LIN {X 0,Y 365.856,Z 163.635,A -85,B 0,C 180,E1 -13024.033,E2 -13024.033} C_VEL
LIN {X 0,Y 364.238,Z 181.611,A -85,B 0,C 180,E1 -13027.845,E2 -13027.845} C_VEL
LIN {X 0,Y 364.107,Z 184.215,A -85,B 0,C 180,E1 -13028.356,E2 -13028.356} C_VEL
LIN {X 0,Y 369.085,Z 220.666,A -85,B 0,C 180,E1 -13029.411,E2 -13029.411} C_VEL
LIN {X 0,Y 367.83,Z 293.633,A -85,B 0,C 180,E1 -13030.937,E2 -13030.937} C_VEL
LIN {X 0,Y 367.143,Z 307.184,A -85,B 0,C 180,E1 -13031.443,E2 -13031.443} C_VEL
LIN {X 0,Y 366.249,Z 319.505,A -85,B 0,C 180,E1 -13032.12,E2 -13032.12} C_VEL
LIN {X 0,Y 365.195,Z 332.175,A -85,B 0,C 180,E1 -13033.078,E2 -13033.078} C_VEL
LIN {X 0,Y 364.123,Z 343.479,A -85,B 0,C 180,E1 -13034.179,E2 -13034.179} C_VEL
LIN {X 0,Y 363.21,Z 353.677,A -85,B 0,C 180,E1 -13035.431,E2 -13035.431} C_VEL
LIN {X 0,Y 362.33,Z 362.875,A -85,B 0,C 180,E1 -13036.826,E2 -13036.826} C_VEL
LIN {X 0,Y 361.664,Z 370.474,A -85,B 0,C 180,E1 -13038.227,E2 -13038.227} C_VEL
LIN {X 0,Y 361.049,Z 377.925,A -85,B 0,C 180,E1 -13039.91,E2 -13039.91} C_VEL
LIN {X 0,Y 360.671,Z 383.894,A -85,B 0,C 180,E1 -13041.596,E2 -13041.596} C_VEL
LIN {X 0,Y 360.485,Z 388.587,A -85,B 0,C 180,E1 -13043.282,E2 -13043.282} C_VEL
LIN {X 0,Y 360.383,Z 392.138,A -85,B 0,C 180,E1 -13044.965,E2 -13044.965} C_VEL
LIN {X 0,Y 360.391,Z 394.652,A -85,B 0,C 180,E1 -13046.646,E2 -13046.646} C_VEL
LIN {X 0,Y 360.472,Z 395.803,A -85,B 0,C 180,E1 -13047.765,E2 -13047.765} C_VEL
LIN {X 0,Y 360.534,Z 396.505,A -85,B 0,C 180,E1 -13048.883,E2 -13048.883} C_VEL
LIN {X 0,Y 360.52,Z 396.804,A -85,B 0,C 180,E1 -13050,E2 -13050} C_VEL
LIN {X 0,Y 360.522,Z 396.707,A -85,B 0,C 180,E1 -13051.117,E2 -13051.117} C_VEL
LIN {X 0,Y 360.428,Z 396.188,A -85,B 0,C 180,E1 -13052.235,E2 -13052.235} C_VEL
LIN {X 0,Y 360.403,Z 393.878,A -85,B 0,C 180,E1 -13054.474,E2 -13054.474} C_VEL
LIN {X 0,Y 360.378,Z 391.416,A -85,B 0,C 180,E1 -13055.961,E2 -13055.961} C_VEL
LIN {X 0,Y 360.596,Z 387.143,A -85,B 0,C 180,E1 -13057.841,E2 -13057.841} C_VEL
LIN {X 0,Y 360.914,Z 382.124,A -85,B 0,C 180,E1 -13059.527,E2 -13059.527} C_VEL
LIN {X 0,Y 361.455,Z 375.833,A -85,B 0,C 180,E1 -13061.212,E2 -13061.212} C_VEL
LIN {X 0,Y 362.392,Z 368.049,A -85,B 0,C 180,E1 -13062.887,E2 -13062.887} C_VEL
LIN {X 0,Y 363.271,Z 360.101,A -85,B 0,C 180,E1 -13064.28,E2 -13064.28} C_VEL
LIN {X 0,Y 364.321,Z 350.431,A -85,B 0,C 180,E1 -13065.668,E2 -13065.668} C_VEL
LIN {X 0,Y 365.477,Z 339.745,A -85,B 0,C 180,E1 -13066.909,E2 -13066.909} C_VEL
LIN {X 0,Y 366.789,Z 327.812,A -85,B 0,C 180,E1 -13067.997,E2 -13067.997} C_VEL
LIN {X 0,Y 367.96,Z 315.104,A -85,B 0,C 180,E1 -13068.875,E2 -13068.875} C_VEL
LIN {X 0,Y 368.927,Z 302.489,A -85,B 0,C 180,E1 -13069.51,E2 -13069.51} C_VEL
LIN {X 0,Y 369.584,Z 289.242,A -85,B 0,C 180,E1 -13069.944,E2 -13069.944} C_VEL
LIN {X 0,Y 370.844,Z 219.661,A -85,B 0,C 180,E1 -13071.411,E2 -13071.411} C_VEL
LIN {X 0,Y 367.604,Z 196.928,A -85,B 0,C 180,E1 -13072.15,E2 -13072.15} C_VEL
LIN {X 0,Y 364.788,Z 182.019,A -85,B 0,C 180,E1 -13072.701,E2 -13072.701} C_VEL
LIN {X 0,Y 366.272,Z 167.518,A -85,B 0,C 180,E1 -13075.777,E2 -13075.777} C_VEL
LIN {X 0,Y 366.461,Z 164.278,A -85,B 0,C 180,E1 -13076.48,E2 -13076.48} C_VEL
LIN {X 0,Y 364.559,Z 154.623,A -85,B 0,C 180,E1 -13078.813,E2 -13078.813} C_VEL
LIN {X 0,Y 361.909,Z 143.406,A -85,B 0,C 180,E1 -13081.704,E2 -13081.704} C_VEL
LIN {X 0,Y 361.869,Z 143.411,A -85,B 0,C 180,E1 -13085.636,E2 -13085.636} C_VEL
LIN {X 0,Y 361.875,Z 143.411,A -85,B 0,C 180,E1 -13089.027,E2 -13089.027} C_VEL
LIN {X 0,Y 361.857,Z 143.415,A -85,B 0,C 180,E1 -13092.435,E2 -13092.435} C_VEL
LIN {X 0,Y 361.826,Z 143.416,A -85,B 0,C 180,E1 -13095.945,E2 -13095.945} C_VEL
LIN {X 0,Y 361.872,Z 143.408,A -85,B 0,C 180,E1 -13099.237,E2 -13099.237} C_VEL
LIN {X 0,Y 361.869,Z 143.408,A -85,B 0,C 180,E1 -13102.982,E2 -13102.982} C_VEL
LIN {X 0,Y 361.858,Z 143.406,A -85,B 0,C 180,E1 -13106.63,E2 -13106.63} C_VEL
LIN {X 0,Y 361.874,Z 143.406,A -85,B 0,C 180,E1 -13109.672,E2 -13109.672} C_VEL
LIN {X 0,Y 361.953,Z 143.394,A -85,B 0,C 180,E1 -13113.475,E2 -13113.475} C_VEL
LIN {X 0,Y 361.881,Z 143.402,A -85,B 0,C 180,E1 -13117.144,E2 -13117.144} C_VEL
LIN {X 0,Y 361.919,Z 143.396,A -85,B 0,C 180,E1 -13120.724,E2 -13120.724} C_VEL
LIN {X 0,Y 361.945,Z 143.393,A -85,B 0,C 180,E1 -13124.226,E2 -13124.226} C_VEL
LIN {X 0,Y 361.997,Z 143.391,A -85,B 0,C 180,E1 -13126.528,E2 -13126.528} C_VEL
LIN {X 0,Y 362.03,Z 143.388,A -85,B 0,C 180,E1 -13129.938,E2 -13129.938} C_VEL
LIN {X 0,Y 362.15,Z 143.368,A -85,B 0,C 180,E1 -13132.192,E2 -13132.192} C_VEL
LIN {X 0,Y 362.117,Z 143.377,A -85,B 0,C 180,E1 -13134.431,E2 -13134.431} C_VEL
LIN {X 0,Y 362.281,Z 143.357,A -85,B 0,C 180,E1 -13137.776,E2 -13137.776} C_VEL
LIN {X 0,Y 362.426,Z 143.334,A -85,B 0,C 180,E1 -13140,E2 -13140} C_VEL
LIN {X 0,Y 362.281,Z 143.356,A -85,B 0,C 180,E1 -13142.223,E2 -13142.223} C_VEL
LIN {X 0,Y 362.159,Z 143.37,A -85,B 0,C 180,E1 -13146.686,E2 -13146.686} C_VEL
LIN {X 0,Y 362.029,Z 143.389,A -85,B 0,C 180,E1 -13150.062,E2 -13150.062} C_VEL
LIN {X 0,Y 361.996,Z 143.391,A -85,B 0,C 180,E1 -13153.899,E2 -13153.899} C_VEL
LIN {X 0,Y 361.965,Z 143.397,A -85,B 0,C 180,E1 -13157.938,E2 -13157.938} C_VEL
LIN {X 0,Y 361.89,Z 143.406,A -85,B 0,C 180,E1 -13161.653,E2 -13161.653} C_VEL
LIN {X 0,Y 361.926,Z 143.407,A -85,B 0,C 180,E1 -13165.29,E2 -13165.29} C_VEL
LIN {X 0,Y 361.93,Z 143.475,A -85,B 0,C 180,E1 -13168.883,E2 -13168.883} C_VEL
LIN {X 0,Y 362.983,Z 148.175,A -85,B 0,C 180,E1 -13170.225,E2 -13170.225} C_VEL
LIN {X 0,Y 370.942,Z 167.193,A -85,B 0,C 180,E1 -13171.263,E2 -13171.263} C_VEL
LIN {X 0,Y 371.99,Z 171.078,A -85,B 0,C 180,E1 -13171.427,E2 -13171.427} C_VEL
LIN {X 0,Y 370.044,Z 255.779,A -85,B 0,C 180,E1 -13173.22,E2 -13173.22} C_VEL
LIN {X 0,Y 369.483,Z 268.943,A -85,B 0,C 180,E1 -13173.723,E2 -13173.723} C_VEL
LIN {X 0,Y 368.876,Z 280.401,A -85,B 0,C 180,E1 -13174.362,E2 -13174.362} C_VEL
LIN {X 0,Y 368.043,Z 291.787,A -85,B 0,C 180,E1 -13175.201,E2 -13175.201} C_VEL
LIN {X 0,Y 366.955,Z 303.498,A -85,B 0,C 180,E1 -13176.32,E2 -13176.32} C_VEL
LIN {X 0,Y 365.859,Z 314.056,A -85,B 0,C 180,E1 -13177.592,E2 -13177.592} C_VEL
LIN {X 0,Y 364.797,Z 323.086,A -85,B 0,C 180,E1 -13178.937,E2 -13178.937} C_VEL
LIN {X 0,Y 363.599,Z 332.307,A -85,B 0,C 180,E1 -13180.654,E2 -13180.654} C_VEL
LIN {X 0,Y 362.718,Z 338.973,A -85,B 0,C 180,E1 -13182.198,E2 -13182.198} C_VEL
LIN {X 0,Y 361.961,Z 345.413,A -85,B 0,C 180,E1 -13184.077,E2 -13184.077} C_VEL
LIN {X 0,Y 361.32,Z 350.44,A -85,B 0,C 180,E1 -13186.028,E2 -13186.028} C_VEL
LIN {X 0,Y 360.911,Z 353.66,A -85,B 0,C 180,E1 -13187.729,E2 -13187.729} C_VEL
LIN {X 0,Y 360.497,Z 356.39,A -85,B 0,C 180,E1 -13189.959,E2 -13189.959} C_VEL
LIN {X 0,Y 360.413,Z 357.239,A -85,B 0,C 180,E1 -13191.392,E2 -13191.392} C_VEL
LIN {X 0,Y 360.34,Z 357.426,A -85,B 0,C 180,E1 -13193.097,E2 -13193.097} C_VEL
LIN {X 0,Y 360.388,Z 356.541,A -85,B 0,C 180,E1 -13194.989,E2 -13194.989} C_VEL
LIN {X 0,Y 360.584,Z 354.422,A -85,B 0,C 180,E1 -13196.939,E2 -13196.939} C_VEL
LIN {X 0,Y 360.927,Z 350.862,A -85,B 0,C 180,E1 -13198.956,E2 -13198.956} C_VEL
LIN {X 0,Y 361.405,Z 345.506,A -85,B 0,C 180,E1 -13201.055,E2 -13201.055} C_VEL
LIN {X 0,Y 361.952,Z 339.784,A -85,B 0,C 180,E1 -13202.761,E2 -13202.761} C_VEL
LIN {X 0,Y 362.663,Z 332.625,A -85,B 0,C 180,E1 -13204.458,E2 -13204.458} C_VEL
LIN {X 0,Y 363.496,Z 324.252,A -85,B 0,C 180,E1 -13206.045,E2 -13206.045} C_VEL
LIN {X 0,Y 364.462,Z 314.352,A -85,B 0,C 180,E1 -13207.561,E2 -13207.561} C_VEL
LIN {X 0,Y 365.415,Z 303.701,A -85,B 0,C 180,E1 -13208.862,E2 -13208.862} C_VEL
LIN {X 0,Y 366.4,Z 291.564,A -85,B 0,C 180,E1 -13210.031,E2 -13210.031} C_VEL
LIN {X 0,Y 367.136,Z 279.291,A -85,B 0,C 180,E1 -13210.941,E2 -13210.941} C_VEL
LIN {X 0,Y 367.783,Z 265.953,A -85,B 0,C 180,E1 -13211.657,E2 -13211.657} C_VEL
LIN {X 0,Y 368.21,Z 253.401,A -85,B 0,C 180,E1 -13212.111,E2 -13212.111} C_VEL
LIN {X 0,Y 369.689,Z 169.162,A -85,B 0,C 180,E1 -13213.858,E2 -13213.858} C_VEL
LIN {X 0,Y 367.562,Z 160.789,A -85,B 0,C 180,E1 -13214.153,E2 -13214.153} C_VEL
LIN {X 0,Y 362.572,Z 146.411,A -85,B 0,C 180,E1 -13214.766,E2 -13214.766} C_VEL
LIN {X 0,Y 361.989,Z 143.397,A -85,B 0,C 180,E1 -13215.609,E2 -13215.609} C_VEL
LIN {X 0,Y 361.969,Z 143.393,A -85,B 0,C 180,E1 -13218.804,E2 -13218.804} C_VEL
LIN {X 0,Y 362.116,Z 143.376,A -85,B 0,C 180,E1 -13222.192,E2 -13222.192} C_VEL
LIN {X 0,Y 362.114,Z 143.375,A -85,B 0,C 180,E1 -13224.431,E2 -13224.431} C_VEL
LIN {X 0,Y 362.28,Z 143.357,A -85,B 0,C 180,E1 -13227.777,E2 -13227.777} C_VEL
LIN {X 0,Y 362.426,Z 143.337,A -85,B 0,C 180,E1 -13230,E2 -13230} C_VEL
LIN {X 0,Y 362.281,Z 143.354,A -85,B 0,C 180,E1 -13232.224,E2 -13232.224} C_VEL
LIN {X 0,Y 362.135,Z 143.374,A -85,B 0,C 180,E1 -13236.687,E2 -13236.687} C_VEL
LIN {X 0,Y 362.048,Z 143.386,A -85,B 0,C 180,E1 -13238.779,E2 -13238.779} C_VEL
LIN {X 0,Y 361.353,Z 143.477,A -85,B 0,C 180,E1 -13239.706,E2 -13239.706} C_VEL
LIN {X 0,Y 358.436,Z 143.838,A -85,B 0,C 180,E1 -13241.214,E2 -13241.214} C_VEL
LIN {X 0,Y 356.005,Z 144.137,A -85,B 0,C 180,E1 -13242.433,E2 -13242.433} C_VEL
LIN {X 0,Y 355.005,Z 144.263,A -85,B 0,C 180,E1 -13243.378,E2 -13243.378} C_VEL
LIN {X 0,Y 354.947,Z 144.268,A -85,B 0,C 180,E1 -13243.698,E2 -13243.698} C_VEL
LIN {X 0,Y 354.879,Z 144.279,A -85,B 0,C 180,E1 -13247.281,E2 -13247.281} C_VEL
LIN {X 0,Y 354.826,Z 144.289,A -85,B 0,C 180,E1 -13250.887,E2 -13250.887} C_VEL
LIN {X 0,Y 354.859,Z 144.283,A -85,B 0,C 180,E1 -13254.576,E2 -13254.576} C_VEL
LIN {X 0,Y 354.883,Z 144.278,A -85,B 0,C 180,E1 -13257.096,E2 -13257.096} C_VEL
LIN {X 0,Y 354.853,Z 144.28,A -85,B 0,C 180,E1 -13259.678,E2 -13259.678} C_VEL
LIN {X 0,Y 354.805,Z 144.286,A -85,B 0,C 180,E1 -13263.702,E2 -13263.702} C_VEL
LIN {X 0,Y 354.797,Z 144.293,A -85,B 0,C 180,E1 -13266.459,E2 -13266.459} C_VEL
LIN {X 0,Y 354.823,Z 144.283,A -85,B 0,C 180,E1 -13269.424,E2 -13269.424} C_VEL
LIN {X 0,Y 354.786,Z 144.289,A -85,B 0,C 180,E1 -13272.867,E2 -13272.867} C_VEL
LIN {X 0,Y 354.766,Z 144.296,A -85,B 0,C 180,E1 -13276.104,E2 -13276.104} C_VEL
LIN {X 0,Y 354.787,Z 144.288,A -85,B 0,C 180,E1 -13279.179,E2 -13279.179} C_VEL
LIN {X 0,Y 354.807,Z 144.288,A -85,B 0,C 180,E1 -13282.402,E2 -13282.402} C_VEL
LIN {X 0,Y 354.811,Z 144.285,A -85,B 0,C 180,E1 -13284.941,E2 -13284.941} C_VEL
LIN {X 0,Y 354.792,Z 144.289,A -85,B 0,C 180,E1 -13288.405,E2 -13288.405} C_VEL
LIN {X 0,Y 354.849,Z 144.284,A -85,B 0,C 180,E1 -13291.619,E2 -13291.619} C_VEL
LIN {X 0,Y 354.897,Z 144.276,A -85,B 0,C 180,E1 -13294.173,E2 -13294.173} C_VEL
LIN {X 0,Y 354.814,Z 144.288,A -85,B 0,C 180,E1 -13297.893,E2 -13297.893} C_VEL
LIN {X 0,Y 354.921,Z 144.274,A -85,B 0,C 180,E1 -13301.891,E2 -13301.891} C_VEL
LIN {X 0,Y 354.941,Z 144.27,A -85,B 0,C 180,E1 -13305.981,E2 -13305.981} C_VEL
LIN {X 0,Y 354.977,Z 144.267,A -85,B 0,C 180,E1 -13309.736,E2 -13309.736} C_VEL
LIN {X 0,Y 355.113,Z 144.248,A -85,B 0,C 180,E1 -13312.037,E2 -13312.037} C_VEL
LIN {X 0,Y 355.091,Z 144.25,A -85,B 0,C 180,E1 -13314.321,E2 -13314.321} C_VEL
LIN {X 0,Y 355.244,Z 144.232,A -85,B 0,C 180,E1 -13317.733,E2 -13317.733} C_VEL
LIN {X 0,Y 355.396,Z 144.212,A -85,B 0,C 180,E1 -13320,E2 -13320} C_VEL
LIN {X 0,Y 355.244,Z 144.231,A -85,B 0,C 180,E1 -13322.268,E2 -13322.268} C_VEL
LIN {X 0,Y 355.124,Z 144.251,A -85,B 0,C 180,E1 -13326.82,E2 -13326.82} C_VEL
LIN {X 0,Y 354.977,Z 144.265,A -85,B 0,C 180,E1 -13330.264,E2 -13330.264} C_VEL
LIN {X 0,Y 354.942,Z 144.269,A -85,B 0,C 180,E1 -13334.019,E2 -13334.019} C_VEL
LIN {X 0,Y 354.922,Z 144.272,A -85,B 0,C 180,E1 -13338.109,E2 -13338.109} C_VEL
LIN {X 0,Y 354.816,Z 144.286,A -85,B 0,C 180,E1 -13342.108,E2 -13342.108} C_VEL
LIN {X 0,Y 354.898,Z 144.275,A -85,B 0,C 180,E1 -13345.828,E2 -13345.828} C_VEL
LIN {X 0,Y 354.853,Z 144.28,A -85,B 0,C 180,E1 -13349.679,E2 -13349.679} C_VEL
LIN {X 0,Y 354.806,Z 144.287,A -85,B 0,C 180,E1 -13353.702,E2 -13353.702} C_VEL
LIN {X 0,Y 354.8,Z 144.29,A -85,B 0,C 180,E1 -13356.46,E2 -13356.46} C_VEL
LIN {X 0,Y 354.824,Z 144.284,A -85,B 0,C 180,E1 -13359.424,E2 -13359.424} C_VEL
LIN {X 0,Y 354.805,Z 144.286,A -85,B 0,C 180,E1 -13362.87,E2 -13362.87} C_VEL
LIN {X 0,Y 354.805,Z 144.286,A -85,B 0,C 180,E1 -13367.13,E2 -13367.13} C_VEL
LIN {X 0,Y 354.838,Z 144.282,A -85,B 0,C 180,E1 -13370.669,E2 -13370.669} C_VEL
LIN {X 0,Y 354.824,Z 144.285,A -85,B 0,C 180,E1 -13374.301,E2 -13374.301} C_VEL
LIN {X 0,Y 354.789,Z 144.294,A -85,B 0,C 180,E1 -13377.667,E2 -13377.667} C_VEL
LIN {X 0,Y 354.829,Z 144.322,A -85,B 0,C 180,E1 -13378.95,E2 -13378.95} C_VEL
LIN {X 0,Y 357.708,Z 157.357,A -85,B 0,C 180,E1 -13382.145,E2 -13382.145} C_VEL
LIN {X 0,Y 358.912,Z 164.923,A -85,B 0,C 180,E1 -13383.92,E2 -13383.92} C_VEL
LIN {X 0,Y 357.173,Z 183.578,A -85,B 0,C 180,E1 -13387.952,E2 -13387.952} C_VEL
LIN {X 0,Y 362.314,Z 220.923,A -85,B 0,C 180,E1 -13389.068,E2 -13389.068} C_VEL
LIN {X 0,Y 361.062,Z 292.895,A -85,B 0,C 180,E1 -13390.603,E2 -13390.603} C_VEL
LIN {X 0,Y 360.387,Z 305.799,A -85,B 0,C 180,E1 -13391.082,E2 -13391.082} C_VEL
LIN {X 0,Y 359.46,Z 318.394,A -85,B 0,C 180,E1 -13391.771,E2 -13391.771} C_VEL
LIN {X 0,Y 358.554,Z 329.68,A -85,B 0,C 180,E1 -13392.608,E2 -13392.608} C_VEL
LIN {X 0,Y 357.361,Z 341.36,A -85,B 0,C 180,E1 -13393.725,E2 -13393.725} C_VEL
LIN {X 0,Y 356.405,Z 351.909,A -85,B 0,C 180,E1 -13395,E2 -13395} C_VEL
LIN {X 0,Y 355.582,Z 360.533,A -85,B 0,C 180,E1 -13396.28,E2 -13396.28} C_VEL
LIN {X 0,Y 354.816,Z 368.48,A -85,B 0,C 180,E1 -13397.706,E2 -13397.706} C_VEL
LIN {X 0,Y 354.06,Z 376.22,A -85,B 0,C 180,E1 -13399.42,E2 -13399.42} C_VEL
LIN {X 0,Y 353.615,Z 383.363,A -85,B 0,C 180,E1 -13401.428,E2 -13401.428} C_VEL
LIN {X 0,Y 353.396,Z 388.087,A -85,B 0,C 180,E1 -13403.147,E2 -13403.147} C_VEL
LIN {X 0,Y 353.289,Z 391.667,A -85,B 0,C 180,E1 -13404.864,E2 -13404.864} C_VEL
LIN {X 0,Y 353.308,Z 394.209,A -85,B 0,C 180,E1 -13406.579,E2 -13406.579} C_VEL
LIN {X 0,Y 353.374,Z 395.381,A -85,B 0,C 180,E1 -13407.72,E2 -13407.72} C_VEL
LIN {X 0,Y 353.468,Z 396.099,A -85,B 0,C 180,E1 -13408.861,E2 -13408.861} C_VEL
LIN {X 0,Y 353.455,Z 396.409,A -85,B 0,C 180,E1 -13410,E2 -13410} C_VEL
LIN {X 0,Y 353.437,Z 396.321,A -85,B 0,C 180,E1 -13411.139,E2 -13411.139} C_VEL
LIN {X 0,Y 353.33,Z 395.821,A -85,B 0,C 180,E1 -13412.28,E2 -13412.28} C_VEL
LIN {X 0,Y 353.286,Z 394.878,A -85,B 0,C 180,E1 -13413.421,E2 -13413.421} C_VEL
LIN {X 0,Y 353.309,Z 393.532,A -85,B 0,C 180,E1 -13414.564,E2 -13414.564} C_VEL
LIN {X 0,Y 353.276,Z 391.434,A -85,B 0,C 180,E1 -13415.905,E2 -13415.905} C_VEL
LIN {X 0,Y 353.526,Z 386.851,A -85,B 0,C 180,E1 -13417.999,E2 -13417.999} C_VEL
LIN {X 0,Y 353.895,Z 381.868,A -85,B 0,C 180,E1 -13419.718,E2 -13419.718} C_VEL
LIN {X 0,Y 354.453,Z 375.613,A -85,B 0,C 180,E1 -13421.436,E2 -13421.436} C_VEL
LIN {X 0,Y 355.45,Z 367.871,A -85,B 0,C 180,E1 -13423.143,E2 -13423.143} C_VEL
LIN {X 0,Y 356.375,Z 359.975,A -85,B 0,C 180,E1 -13424.563,E2 -13424.563} C_VEL
LIN {X 0,Y 357.465,Z 350.362,A -85,B 0,C 180,E1 -13425.977,E2 -13425.977} C_VEL
LIN {X 0,Y 358.682,Z 339.741,A -85,B 0,C 180,E1 -13427.239,E2 -13427.239} C_VEL
LIN {X 0,Y 360.055,Z 327.947,A -85,B 0,C 180,E1 -13428.345,E2 -13428.345} C_VEL
LIN {X 0,Y 361.263,Z 315.396,A -85,B 0,C 180,E1 -13429.238,E2 -13429.238} C_VEL
LIN {X 0,Y 362.31,Z 302.274,A -85,B 0,C 180,E1 -13429.918,E2 -13429.918} C_VEL
LIN {X 0,Y 363.018,Z 289.279,A -85,B 0,C 180,E1 -13430.357,E2 -13430.357} C_VEL
LIN {X 0,Y 364.398,Z 220.897,A -85,B 0,C 180,E1 -13431.83,E2 -13431.83} C_VEL
LIN {X 0,Y 361.153,Z 198.061,A -85,B 0,C 180,E1 -13432.596,E2 -13432.596} C_VEL
LIN {X 0,Y 358.058,Z 181.553,A -85,B 0,C 180,E1 -13433.228,E2 -13433.228} C_VEL
LIN {X 0,Y 359.626,Z 166.696,A -85,B 0,C 180,E1 -13436.454,E2 -13436.454} C_VEL
LIN {X 0,Y 358.255,Z 158.685,A -85,B 0,C 180,E1 -13438.405,E2 -13438.405} C_VEL
LIN {X 0,Y 355.259,Z 145.919,A -85,B 0,C 180,E1 -13441.716,E2 -13441.716} C_VEL
LIN {X 0,Y 354.839,Z 144.287,A -85,B 0,C 180,E1 -13442.227,E2 -13442.227} C_VEL
LIN {X 0,Y 354.823,Z 144.289,A -85,B 0,C 180,E1 -13445.699,E2 -13445.699} C_VEL
LIN {X 0,Y 354.825,Z 144.29,A -85,B 0,C 180,E1 -13449.423,E2 -13449.423} C_VEL
LIN {X 0,Y 354.805,Z 144.291,A -85,B 0,C 180,E1 -13452.87,E2 -13452.87} C_VEL
LIN {X 0,Y 354.804,Z 144.291,A -85,B 0,C 180,E1 -13457.13,E2 -13457.13} C_VEL
LIN {X 0,Y 354.837,Z 144.281,A -85,B 0,C 180,E1 -13460.669,E2 -13460.669} C_VEL
LIN {X 0,Y 354.822,Z 144.284,A -85,B 0,C 180,E1 -13464.3,E2 -13464.3} C_VEL
LIN {X 0,Y 354.786,Z 144.288,A -85,B 0,C 180,E1 -13467.666,E2 -13467.666} C_VEL
LIN {X 0,Y 354.868,Z 144.274,A -85,B 0,C 180,E1 -13470.621,E2 -13470.621} C_VEL
LIN {X 0,Y 354.898,Z 144.271,A -85,B 0,C 180,E1 -13474.172,E2 -13474.172} C_VEL
LIN {X 0,Y 354.815,Z 144.282,A -85,B 0,C 180,E1 -13477.892,E2 -13477.892} C_VEL
LIN {X 0,Y 354.922,Z 144.27,A -85,B 0,C 180,E1 -13481.891,E2 -13481.891} C_VEL
LIN {X 0,Y 354.941,Z 144.27,A -85,B 0,C 180,E1 -13485.981,E2 -13485.981} C_VEL
LIN {X 0,Y 354.976,Z 144.267,A -85,B 0,C 180,E1 -13489.736,E2 -13489.736} C_VEL
LIN {X 0,Y 355.113,Z 144.244,A -85,B 0,C 180,E1 -13492.037,E2 -13492.037} C_VEL
LIN {X 0,Y 355.091,Z 144.252,A -85,B 0,C 180,E1 -13494.32,E2 -13494.32} C_VEL
LIN {X 0,Y 355.244,Z 144.234,A -85,B 0,C 180,E1 -13497.732,E2 -13497.732} C_VEL
LIN {X 0,Y 355.396,Z 144.21,A -85,B 0,C 180,E1 -13500,E2 -13500} C_VEL
LIN {X 0,Y 355.244,Z 144.233,A -85,B 0,C 180,E1 -13502.267,E2 -13502.267} C_VEL
LIN {X 0,Y 355.122,Z 144.248,A -85,B 0,C 180,E1 -13506.819,E2 -13506.819} C_VEL
LIN {X 0,Y 354.976,Z 144.268,A -85,B 0,C 180,E1 -13510.264,E2 -13510.264} C_VEL
LIN {X 0,Y 354.94,Z 144.27,A -85,B 0,C 180,E1 -13514.019,E2 -13514.019} C_VEL
LIN {X 0,Y 354.921,Z 144.274,A -85,B 0,C 180,E1 -13518.109,E2 -13518.109} C_VEL
LIN {X 0,Y 354.833,Z 144.288,A -85,B 0,C 180,E1 -13522.106,E2 -13522.106} C_VEL
LIN {X 0,Y 354.897,Z 144.28,A -85,B 0,C 180,E1 -13525.827,E2 -13525.827} C_VEL
LIN {X 0,Y 354.902,Z 144.37,A -85,B 0,C 180,E1 -13528.415,E2 -13528.415} C_VEL
LIN {X 0,Y 355.876,Z 148.704,A -85,B 0,C 180,E1 -13529.666,E2 -13529.666} C_VEL
LIN {X 0,Y 363.7,Z 166.992,A -85,B 0,C 180,E1 -13530.721,E2 -13530.721} C_VEL
LIN {X 0,Y 365.427,Z 171.738,A -85,B 0,C 180,E1 -13530.961,E2 -13530.961} C_VEL
LIN {X 0,Y 363.518,Z 255.538,A -85,B 0,C 180,E1 -13532.774,E2 -13532.774} C_VEL
LIN {X 0,Y 362.94,Z 268.373,A -85,B 0,C 180,E1 -13533.26,E2 -13533.26} C_VEL
LIN {X 0,Y 362.299,Z 280.563,A -85,B 0,C 180,E1 -13533.945,E2 -13533.945} C_VEL
LIN {X 0,Y 361.372,Z 292.386,A -85,B 0,C 180,E1 -13534.831,E2 -13534.831} C_VEL
LIN {X 0,Y 360.278,Z 303.61,A -85,B 0,C 180,E1 -13535.922,E2 -13535.922} C_VEL
LIN {X 0,Y 359.233,Z 313.375,A -85,B 0,C 180,E1 -13537.105,E2 -13537.105} C_VEL
LIN {X 0,Y 358.018,Z 323.206,A -85,B 0,C 180,E1 -13538.569,E2 -13538.569} C_VEL
LIN {X 0,Y 356.785,Z 332.224,A -85,B 0,C 180,E1 -13540.262,E2 -13540.262} C_VEL
LIN {X 0,Y 355.831,Z 339.067,A -85,B 0,C 180,E1 -13541.858,E2 -13541.858} C_VEL
LIN {X 0,Y 355.136,Z 344.609,A -85,B 0,C 180,E1 -13543.46,E2 -13543.46} C_VEL
LIN {X 0,Y 354.503,Z 349.067,A -85,B 0,C 180,E1 -13545.07,E2 -13545.07} C_VEL
LIN {X 0,Y 354.06,Z 352.562,A -85,B 0,C 180,E1 -13546.697,E2 -13546.697} C_VEL
LIN {X 0,Y 353.889,Z 353.989,A -85,B 0,C 180,E1 -13547.529,E2 -13547.529} C_VEL
LIN {X 0,Y 353.553,Z 356.033,A -85,B 0,C 180,E1 -13549.057,E2 -13549.057} C_VEL
LIN {X 0,Y 353.321,Z 357.467,A -85,B 0,C 180,E1 -13550.874,E2 -13550.874} C_VEL
LIN {X 0,Y 353.273,Z 357.875,A -85,B 0,C 180,E1 -13552.727,E2 -13552.727} C_VEL
LIN {X 0,Y 353.281,Z 357.092,A -85,B 0,C 180,E1 -13554.767,E2 -13554.767} C_VEL
LIN {X 0,Y 353.458,Z 355.263,A -85,B 0,C 180,E1 -13556.627,E2 -13556.627} C_VEL
LIN {X 0,Y 353.798,Z 351.966,A -85,B 0,C 180,E1 -13558.668,E2 -13558.668} C_VEL
LIN {X 0,Y 354.265,Z 346.961,A -85,B 0,C 180,E1 -13560.795,E2 -13560.795} C_VEL
LIN {X 0,Y 354.794,Z 341.351,A -85,B 0,C 180,E1 -13562.578,E2 -13562.578} C_VEL
LIN {X 0,Y 355.621,Z 333.626,A -85,B 0,C 180,E1 -13564.502,E2 -13564.502} C_VEL
LIN {X 0,Y 356.482,Z 325.164,A -85,B 0,C 180,E1 -13566.162,E2 -13566.162} C_VEL
LIN {X 0,Y 357.376,Z 316.39,A -85,B 0,C 180,E1 -13567.56,E2 -13567.56} C_VEL
LIN {X 0,Y 358.315,Z 306.269,A -85,B 0,C 180,E1 -13568.875,E2 -13568.875} C_VEL
LIN {X 0,Y 359.304,Z 295.223,A -85,B 0,C 180,E1 -13570.021,E2 -13570.021} C_VEL
LIN {X 0,Y 360.136,Z 283.2,A -85,B 0,C 180,E1 -13570.995,E2 -13570.995} C_VEL
LIN {X 0,Y 360.826,Z 270.514,A -85,B 0,C 180,E1 -13571.769,E2 -13571.769} C_VEL
LIN {X 0,Y 361.274,Z 258.092,A -85,B 0,C 180,E1 -13572.296,E2 -13572.296} C_VEL
LIN {X 0,Y 361.697,Z 241.624,A -85,B 0,C 180,E1 -13572.703,E2 -13572.703} C_VEL
LIN {X 0,Y 363.015,Z 170.323,A -85,B 0,C 180,E1 -13574.193,E2 -13574.193} C_VEL
LIN {X 0,Y 361.18,Z 163.241,A -85,B 0,C 180,E1 -13574.451,E2 -13574.451} C_VEL
LIN {X 0,Y 355.43,Z 146.758,A -85,B 0,C 180,E1 -13575.172,E2 -13575.172} C_VEL
LIN {X 0,Y 354.977,Z 144.27,A -85,B 0,C 180,E1 -13575.89,E2 -13575.89} C_VEL
LIN {X 0,Y 354.977,Z 144.269,A -85,B 0,C 180,E1 -13579.736,E2 -13579.736} C_VEL
LIN {X 0,Y 355.124,Z 144.249,A -85,B 0,C 180,E1 -13583.181,E2 -13583.181} C_VEL
LIN {X 0,Y 355.243,Z 144.234,A -85,B 0,C 180,E1 -13587.732,E2 -13587.732} C_VEL
LIN {X 0,Y 355.396,Z 144.213,A -85,B 0,C 180,E1 -13590,E2 -13590} C_VEL
LIN {X 0,Y 355.244,Z 144.231,A -85,B 0,C 180,E1 -13592.268,E2 -13592.268} C_VEL
LIN {X 0,Y 355.099,Z 144.252,A -85,B 0,C 180,E1 -13596.82,E2 -13596.82} C_VEL
LIN {X 0,Y 354.956,Z 144.267,A -85,B 0,C 180,E1 -13600.265,E2 -13600.265} C_VEL
LIN {X 0,Y 354.947,Z 144.268,A -85,B 0,C 180,E1 -13603.698,E2 -13603.698} C_VEL
LIN {X 0,Y 354.333,Z 144.35,A -85,B 0,C 180,E1 -13604.644,E2 -13604.644} C_VEL
LIN {X 0,Y 351.459,Z 144.703,A -85,B 0,C 180,E1 -13606.182,E2 -13606.182} C_VEL
LIN {X 0,Y 348.977,Z 145.013,A -85,B 0,C 180,E1 -13607.426,E2 -13607.426} C_VEL
LIN {X 0,Y 347.895,Z 145.148,A -85,B 0,C 180,E1 -13608.39,E2 -13608.39} C_VEL
LIN {X 0,Y 347.801,Z 145.162,A -85,B 0,C 180,E1 -13608.717,E2 -13608.717} C_VEL
LIN {X 0,Y 347.763,Z 145.167,A -85,B 0,C 180,E1 -13612.58,E2 -13612.58} C_VEL
LIN {X 0,Y 347.811,Z 145.159,A -85,B 0,C 180,E1 -13615.108,E2 -13615.108} C_VEL
LIN {X 0,Y 347.81,Z 145.157,A -85,B 0,C 180,E1 -13617.694,E2 -13617.694} C_VEL
LIN {X 0,Y 347.763,Z 145.166,A -85,B 0,C 180,E1 -13620.346,E2 -13620.346} C_VEL
LIN {X 0,Y 347.743,Z 145.171,A -85,B 0,C 180,E1 -13624.464,E2 -13624.464} C_VEL
LIN {X 0,Y 347.771,Z 145.164,A -85,B 0,C 180,E1 -13627.988,E2 -13627.988} C_VEL
LIN {X 0,Y 347.749,Z 145.166,A -85,B 0,C 180,E1 -13631.83,E2 -13631.83} C_VEL
LIN {X 0,Y 347.705,Z 145.17,A -85,B 0,C 180,E1 -13635.027,E2 -13635.027} C_VEL
LIN {X 0,Y 347.749,Z 145.168,A -85,B 0,C 180,E1 -13638.397,E2 -13638.397} C_VEL
LIN {X 0,Y 347.773,Z 145.167,A -85,B 0,C 180,E1 -13642.011,E2 -13642.011} C_VEL
LIN {X 0,Y 347.743,Z 145.167,A -85,B 0,C 180,E1 -13645.536,E2 -13645.536} C_VEL
LIN {X 0,Y 347.762,Z 145.167,A -85,B 0,C 180,E1 -13649.654,E2 -13649.654} C_VEL
LIN {X 0,Y 347.85,Z 145.152,A -85,B 0,C 180,E1 -13652.745,E2 -13652.745} C_VEL
LIN {X 0,Y 347.783,Z 145.162,A -85,B 0,C 180,E1 -13656.162,E2 -13656.162} C_VEL
LIN {X 0,Y 347.81,Z 145.16,A -85,B 0,C 180,E1 -13659.909,E2 -13659.909} C_VEL
LIN {X 0,Y 347.865,Z 145.15,A -85,B 0,C 180,E1 -13662.359,E2 -13662.359} C_VEL
LIN {X 0,Y 347.896,Z 145.148,A -85,B 0,C 180,E1 -13665.971,E2 -13665.971} C_VEL
LIN {X 0,Y 347.927,Z 145.147,A -85,B 0,C 180,E1 -13669.526,E2 -13669.526} C_VEL
LIN {X 0,Y 348.073,Z 145.125,A -85,B 0,C 180,E1 -13671.875,E2 -13671.875} C_VEL
LIN {X 0,Y 348.066,Z 145.125,A -85,B 0,C 180,E1 -13674.206,E2 -13674.206} C_VEL
LIN {X 0,Y 348.206,Z 145.109,A -85,B 0,C 180,E1 -13677.687,E2 -13677.687} C_VEL
LIN {X 0,Y 348.345,Z 145.09,A -85,B 0,C 180,E1 -13680,E2 -13680} C_VEL
LIN {X 0,Y 348.207,Z 145.108,A -85,B 0,C 180,E1 -13682.314,E2 -13682.314} C_VEL
LIN {X 0,Y 348.09,Z 145.128,A -85,B 0,C 180,E1 -13686.958,E2 -13686.958} C_VEL
LIN {X 0,Y 347.928,Z 145.145,A -85,B 0,C 180,E1 -13690.475,E2 -13690.475} C_VEL
LIN {X 0,Y 347.898,Z 145.147,A -85,B 0,C 180,E1 -13694.15,E2 -13694.15} C_VEL
LIN {X 0,Y 347.891,Z 145.149,A -85,B 0,C 180,E1 -13698.291,E2 -13698.291} C_VEL
LIN {X 0,Y 347.767,Z 145.162,A -85,B 0,C 180,E1 -13701.627,E2 -13701.627} C_VEL
LIN {X 0,Y 347.811,Z 145.158,A -85,B 0,C 180,E1 -13705.109,E2 -13705.109} C_VEL
LIN {X 0,Y 347.81,Z 145.157,A -85,B 0,C 180,E1 -13707.694,E2 -13707.694} C_VEL
LIN {X 0,Y 347.763,Z 145.169,A -85,B 0,C 180,E1 -13710.347,E2 -13710.347} C_VEL
LIN {X 0,Y 347.744,Z 145.169,A -85,B 0,C 180,E1 -13714.464,E2 -13714.464} C_VEL
LIN {X 0,Y 347.776,Z 145.166,A -85,B 0,C 180,E1 -13717.99,E2 -13717.99} C_VEL
LIN {X 0,Y 347.767,Z 145.166,A -85,B 0,C 180,E1 -13721.828,E2 -13721.828} C_VEL
LIN {X 0,Y 347.734,Z 145.166,A -85,B 0,C 180,E1 -13725.022,E2 -13725.022} C_VEL
LIN {X 0,Y 347.769,Z 145.164,A -85,B 0,C 180,E1 -13728.394,E2 -13728.394} C_VEL
LIN {X 0,Y 347.777,Z 145.165,A -85,B 0,C 180,E1 -13732.011,E2 -13732.011} C_VEL
LIN {X 0,Y 347.746,Z 145.169,A -85,B 0,C 180,E1 -13735.536,E2 -13735.536} C_VEL
LIN {X 0,Y 347.772,Z 145.277,A -85,B 0,C 180,E1 -13738.643,E2 -13738.643} C_VEL
LIN {X 0,Y 350.813,Z 158.956,A -85,B 0,C 180,E1 -13742.072,E2 -13742.072} C_VEL
LIN {X 0,Y 351.905,Z 165.397,A -85,B 0,C 180,E1 -13743.618,E2 -13743.618} C_VEL
LIN {X 0,Y 350.64,Z 179.139,A -85,B 0,C 180,E1 -13746.657,E2 -13746.657} C_VEL
LIN {X 0,Y 350.284,Z 183.172,A -85,B 0,C 180,E1 -13747.543,E2 -13747.543} C_VEL
LIN {X 0,Y 355.567,Z 222.023,A -85,B 0,C 180,E1 -13748.74,E2 -13748.74} C_VEL
LIN {X 0,Y 354.234,Z 292.995,A -85,B 0,C 180,E1 -13750.289,E2 -13750.289} C_VEL
LIN {X 0,Y 353.53,Z 306.501,A -85,B 0,C 180,E1 -13750.814,E2 -13750.814} C_VEL
LIN {X 0,Y 352.513,Z 319.298,A -85,B 0,C 180,E1 -13751.549,E2 -13751.549} C_VEL
LIN {X 0,Y 351.423,Z 331.855,A -85,B 0,C 180,E1 -13752.544,E2 -13752.544} C_VEL
LIN {X 0,Y 350.27,Z 343.083,A -85,B 0,C 180,E1 -13753.686,E2 -13753.686} C_VEL
LIN {X 0,Y 349.272,Z 353.191,A -85,B 0,C 180,E1 -13754.984,E2 -13754.984} C_VEL
LIN {X 0,Y 348.251,Z 363.184,A -85,B 0,C 180,E1 -13756.58,E2 -13756.58} C_VEL
LIN {X 0,Y 347.537,Z 370.609,A -85,B 0,C 180,E1 -13758.037,E2 -13758.037} C_VEL
LIN {X 0,Y 346.881,Z 377.904,A -85,B 0,C 180,E1 -13759.789,E2 -13759.789} C_VEL
LIN {X 0,Y 346.541,Z 382.819,A -85,B 0,C 180,E1 -13761.251,E2 -13761.251} C_VEL
LIN {X 0,Y 346.321,Z 387.58,A -85,B 0,C 180,E1 -13763.006,E2 -13763.006} C_VEL
LIN {X 0,Y 346.205,Z 390.696,A -85,B 0,C 180,E1 -13764.49,E2 -13764.49} C_VEL
LIN {X 0,Y 346.227,Z 393.762,A -85,B 0,C 180,E1 -13766.509,E2 -13766.509} C_VEL
LIN {X 0,Y 346.277,Z 394.954,A -85,B 0,C 180,E1 -13767.674,E2 -13767.674} C_VEL
LIN {X 0,Y 346.385,Z 395.69,A -85,B 0,C 180,E1 -13768.837,E2 -13768.837} C_VEL
LIN {X 0,Y 346.392,Z 396.013,A -85,B 0,C 180,E1 -13770,E2 -13770} C_VEL
LIN {X 0,Y 346.355,Z 395.936,A -85,B 0,C 180,E1 -13771.163,E2 -13771.163} C_VEL
LIN {X 0,Y 346.232,Z 395.454,A -85,B 0,C 180,E1 -13772.327,E2 -13772.327} C_VEL
LIN {X 0,Y 346.205,Z 394.531,A -85,B 0,C 180,E1 -13773.491,E2 -13773.491} C_VEL
LIN {X 0,Y 346.219,Z 393.198,A -85,B 0,C 180,E1 -13774.657,E2 -13774.657} C_VEL
LIN {X 0,Y 346.224,Z 390.4,A -85,B 0,C 180,E1 -13776.409,E2 -13776.409} C_VEL
LIN {X 0,Y 346.477,Z 386.572,A -85,B 0,C 180,E1 -13778.163,E2 -13778.163} C_VEL
LIN {X 0,Y 346.86,Z 381.617,A -85,B 0,C 180,E1 -13779.917,E2 -13779.917} C_VEL
LIN {X 0,Y 347.466,Z 375.392,A -85,B 0,C 180,E1 -13781.669,E2 -13781.669} C_VEL
LIN {X 0,Y 348.515,Z 367.688,A -85,B 0,C 180,E1 -13783.409,E2 -13783.409} C_VEL
LIN {X 0,Y 349.484,Z 359.839,A -85,B 0,C 180,E1 -13784.856,E2 -13784.856} C_VEL
LIN {X 0,Y 350.614,Z 350.299,A -85,B 0,C 180,E1 -13786.297,E2 -13786.297} C_VEL
LIN {X 0,Y 351.913,Z 339.775,A -85,B 0,C 180,E1 -13787.581,E2 -13787.581} C_VEL
LIN {X 0,Y 353.324,Z 328.129,A -85,B 0,C 180,E1 -13788.708,E2 -13788.708} C_VEL
LIN {X 0,Y 354.589,Z 315.828,A -85,B 0,C 180,E1 -13789.615,E2 -13789.615} C_VEL
LIN {X 0,Y 355.729,Z 302.286,A -85,B 0,C 180,E1 -13790.34,E2 -13790.34} C_VEL
LIN {X 0,Y 356.485,Z 289.691,A -85,B 0,C 180,E1 -13790.785,E2 -13790.785} C_VEL
LIN {X 0,Y 357.905,Z 221.604,A -85,B 0,C 180,E1 -13792.286,E2 -13792.286} C_VEL
LIN {X 0,Y 354.821,Z 199.637,A -85,B 0,C 180,E1 -13793.041,E2 -13793.041} C_VEL
LIN {X 0,Y 351.371,Z 181.037,A -85,B 0,C 180,E1 -13793.791,E2 -13793.791} C_VEL
LIN {X 0,Y 352.786,Z 168.158,A -85,B 0,C 180,E1 -13796.651,E2 -13796.651} C_VEL
LIN {X 0,Y 351.338,Z 159.985,A -85,B 0,C 180,E1 -13798.691,E2 -13798.691} C_VEL
LIN {X 0,Y 348.347,Z 147.309,A -85,B 0,C 180,E1 -13802.074,E2 -13802.074} C_VEL
LIN {X 0,Y 347.769,Z 145.168,A -85,B 0,C 180,E1 -13802.696,E2 -13802.696} C_VEL
LIN {X 0,Y 347.772,Z 145.171,A -85,B 0,C 180,E1 -13806.065,E2 -13806.065} C_VEL
LIN {X 0,Y 347.759,Z 145.173,A -85,B 0,C 180,E1 -13809.829,E2 -13809.829} C_VEL
LIN {X 0,Y 347.73,Z 145.172,A -85,B 0,C 180,E1 -13813.407,E2 -13813.407} C_VEL
LIN {X 0,Y 347.746,Z 145.171,A -85,B 0,C 180,E1 -13816.682,E2 -13816.682} C_VEL
LIN {X 0,Y 347.758,Z 145.167,A -85,B 0,C 180,E1 -13820.17,E2 -13820.17} C_VEL
LIN {X 0,Y 347.771,Z 145.162,A -85,B 0,C 180,E1 -13823.934,E2 -13823.934} C_VEL
LIN {X 0,Y 347.732,Z 145.165,A -85,B 0,C 180,E1 -13826.927,E2 -13826.927} C_VEL
LIN {X 0,Y 347.804,Z 145.154,A -85,B 0,C 180,E1 -13830.99,E2 -13830.99} C_VEL
LIN {X 0,Y 347.83,Z 145.152,A -85,B 0,C 180,E1 -13833.607,E2 -13833.607} C_VEL
LIN {X 0,Y 347.784,Z 145.159,A -85,B 0,C 180,E1 -13836.161,E2 -13836.161} C_VEL
LIN {X 0,Y 347.81,Z 145.155,A -85,B 0,C 180,E1 -13839.909,E2 -13839.909} C_VEL
LIN {X 0,Y 347.865,Z 145.149,A -85,B 0,C 180,E1 -13842.359,E2 -13842.359} C_VEL
LIN {X 0,Y 347.896,Z 145.148,A -85,B 0,C 180,E1 -13845.97,E2 -13845.97} C_VEL
LIN {X 0,Y 347.927,Z 145.143,A -85,B 0,C 180,E1 -13849.525,E2 -13849.525} C_VEL
LIN {X 0,Y 348.073,Z 145.122,A -85,B 0,C 180,E1 -13851.874,E2 -13851.874} C_VEL
LIN {X 0,Y 348.066,Z 145.127,A -85,B 0,C 180,E1 -13854.205,E2 -13854.205} C_VEL
LIN {X 0,Y 348.206,Z 145.111,A -85,B 0,C 180,E1 -13857.686,E2 -13857.686} C_VEL
LIN {X 0,Y 348.344,Z 145.088,A -85,B 0,C 180,E1 -13860,E2 -13860} C_VEL
LIN {X 0,Y 348.206,Z 145.11,A -85,B 0,C 180,E1 -13862.313,E2 -13862.313} C_VEL
LIN {X 0,Y 348.088,Z 145.125,A -85,B 0,C 180,E1 -13866.958,E2 -13866.958} C_VEL
LIN {X 0,Y 347.926,Z 145.148,A -85,B 0,C 180,E1 -13870.474,E2 -13870.474} C_VEL
LIN {X 0,Y 347.896,Z 145.148,A -85,B 0,C 180,E1 -13874.15,E2 -13874.15} C_VEL
LIN {X 0,Y 347.889,Z 145.15,A -85,B 0,C 180,E1 -13878.29,E2 -13878.29} C_VEL
LIN {X 0,Y 347.786,Z 145.163,A -85,B 0,C 180,E1 -13881.635,E2 -13881.635} C_VEL
LIN {X 0,Y 347.81,Z 145.167,A -85,B 0,C 180,E1 -13885.108,E2 -13885.108} C_VEL
LIN {X 0,Y 347.849,Z 145.347,A -85,B 0,C 180,E1 -13887.936,E2 -13887.936} C_VEL
LIN {X 0,Y 348.702,Z 149.035,A -85,B 0,C 180,E1 -13889.052,E2 -13889.052} C_VEL
LIN {X 0,Y 356.591,Z 167.076,A -85,B 0,C 180,E1 -13890.17,E2 -13890.17} C_VEL
LIN {X 0,Y 359.121,Z 173.662,A -85,B 0,C 180,E1 -13890.527,E2 -13890.527} C_VEL
LIN {X 0,Y 357.005,Z 256.112,A -85,B 0,C 180,E1 -13892.336,E2 -13892.336} C_VEL
LIN {X 0,Y 356.389,Z 269.136,A -85,B 0,C 180,E1 -13892.842,E2 -13892.842} C_VEL
LIN {X 0,Y 355.662,Z 282.057,A -85,B 0,C 180,E1 -13893.593,E2 -13893.593} C_VEL
LIN {X 0,Y 354.767,Z 292.824,A -85,B 0,C 180,E1 -13894.426,E2 -13894.426} C_VEL
LIN {X 0,Y 353.669,Z 303.751,A -85,B 0,C 180,E1 -13895.505,E2 -13895.505} C_VEL
LIN {X 0,Y 352.507,Z 313.756,A -85,B 0,C 180,E1 -13896.735,E2 -13896.735} C_VEL
LIN {X 0,Y 351.316,Z 322.83,A -85,B 0,C 180,E1 -13898.103,E2 -13898.103} C_VEL
LIN {X 0,Y 350.085,Z 331.575,A -85,B 0,C 180,E1 -13899.732,E2 -13899.732} C_VEL
LIN {X 0,Y 348.866,Z 339.778,A -85,B 0,C 180,E1 -13901.666,E2 -13901.666} C_VEL
LIN {X 0,Y 348.102,Z 345.505,A -85,B 0,C 180,E1 -13903.38,E2 -13903.38} C_VEL
LIN {X 0,Y 347.452,Z 349.968,A -85,B 0,C 180,E1 -13905.068,E2 -13905.068} C_VEL
LIN {X 0,Y 346.973,Z 353.495,A -85,B 0,C 180,E1 -13906.818,E2 -13906.818} C_VEL
LIN {X 0,Y 346.544,Z 356.078,A -85,B 0,C 180,E1 -13908.622,E2 -13908.622} C_VEL
LIN {X 0,Y 346.272,Z 357.676,A -85,B 0,C 180,E1 -13910.466,E2 -13910.466} C_VEL
LIN {X 0,Y 346.197,Z 358.272,A -85,B 0,C 180,E1 -13912.482,E2 -13912.482} C_VEL
LIN {X 0,Y 346.177,Z 357.769,A -85,B 0,C 180,E1 -13914.298,E2 -13914.298} C_VEL
LIN {X 0,Y 346.311,Z 356.083,A -85,B 0,C 180,E1 -13916.309,E2 -13916.309} C_VEL
LIN {X 0,Y 346.662,Z 353.018,A -85,B 0,C 180,E1 -13918.373,E2 -13918.373} C_VEL
LIN {X 0,Y 347.119,Z 348.319,A -85,B 0,C 180,E1 -13920.529,E2 -13920.529} C_VEL
LIN {X 0,Y 347.598,Z 343.198,A -85,B 0,C 180,E1 -13922.288,E2 -13922.288} C_VEL
LIN {X 0,Y 348.293,Z 337.043,A -85,B 0,C 180,E1 -13923.968,E2 -13923.968} C_VEL
LIN {X 0,Y 349.111,Z 329.49,A -85,B 0,C 180,E1 -13925.626,E2 -13925.626} C_VEL
LIN {X 0,Y 350.09,Z 320.618,A -85,B 0,C 180,E1 -13927.202,E2 -13927.202} C_VEL
LIN {X 0,Y 351.004,Z 311.203,A -85,B 0,C 180,E1 -13928.567,E2 -13928.567} C_VEL
LIN {X 0,Y 351.993,Z 300.813,A -85,B 0,C 180,E1 -13929.787,E2 -13929.787} C_VEL
LIN {X 0,Y 352.897,Z 289.759,A -85,B 0,C 180,E1 -13930.816,E2 -13930.816} C_VEL
LIN {X 0,Y 353.608,Z 277.837,A -85,B 0,C 180,E1 -13931.684,E2 -13931.684} C_VEL
LIN {X 0,Y 354.256,Z 264.885,A -85,B 0,C 180,E1 -13932.372,E2 -13932.372} C_VEL
LIN {X 0,Y 354.71,Z 251.834,A -85,B 0,C 180,E1 -13932.817,E2 -13932.817} C_VEL
LIN {X 0,Y 356.21,Z 170.991,A -85,B 0,C 180,E1 -13934.556,E2 -13934.556} C_VEL
LIN {X 0,Y 354.343,Z 164.36,A -85,B 0,C 180,E1 -13934.813,E2 -13934.813} C_VEL
LIN {X 0,Y 348.319,Z 147.16,A -85,B 0,C 180,E1 -13935.578,E2 -13935.578} C_VEL
LIN {X 0,Y 347.941,Z 145.146,A -85,B 0,C 180,E1 -13936.196,E2 -13936.196} C_VEL
LIN {X 0,Y 347.928,Z 145.148,A -85,B 0,C 180,E1 -13939.526,E2 -13939.526} C_VEL
LIN {X 0,Y 348.09,Z 145.124,A -85,B 0,C 180,E1 -13943.042,E2 -13943.042} C_VEL
LIN {X 0,Y 348.205,Z 145.111,A -85,B 0,C 180,E1 -13947.687,E2 -13947.687} C_VEL
LIN {X 0,Y 348.345,Z 145.091,A -85,B 0,C 180,E1 -13950,E2 -13950} C_VEL
LIN {X 0,Y 348.206,Z 145.108,A -85,B 0,C 180,E1 -13952.314,E2 -13952.314} C_VEL
LIN {X 0,Y 348.064,Z 145.129,A -85,B 0,C 180,E1 -13956.958,E2 -13956.958} C_VEL
LIN {X 0,Y 347.896,Z 145.147,A -85,B 0,C 180,E1 -13960.475,E2 -13960.475} C_VEL
LIN {X 0,Y 347.898,Z 145.146,A -85,B 0,C 180,E1 -13964.15,E2 -13964.15} C_VEL
LIN {X 0,Y 347.828,Z 145.156,A -85,B 0,C 180,E1 -13968.259,E2 -13968.259} C_VEL
LIN {X 0,Y 347.801,Z 145.162,A -85,B 0,C 180,E1 -13968.717,E2 -13968.717} C_VEL
LIN {X 0,Y 347.108,Z 145.255,A -85,B 0,C 180,E1 -13969.683,E2 -13969.683} C_VEL
LIN {X 0,Y 344.221,Z 145.614,A -85,B 0,C 180,E1 -13971.255,E2 -13971.255} C_VEL
LIN {X 0,Y 341.803,Z 145.909,A -85,B 0,C 180,E1 -13972.527,E2 -13972.527} C_VEL
LIN {X 0,Y 340.79,Z 146.032,A -85,B 0,C 180,E1 -13973.512,E2 -13973.512} C_VEL
LIN {X 0,Y 340.72,Z 146.04,A -85,B 0,C 180,E1 -13973.846,E2 -13973.846} C_VEL
LIN {X 0,Y 340.778,Z 146.033,A -85,B 0,C 180,E1 -13977.526,E2 -13977.526} C_VEL
LIN {X 0,Y 340.703,Z 146.044,A -85,B 0,C 180,E1 -13981.044,E2 -13981.044} C_VEL
LIN {X 0,Y 340.717,Z 146.041,A -85,B 0,C 180,E1 -13985.279,E2 -13985.279} C_VEL
LIN {X 0,Y 340.708,Z 146.048,A -85,B 0,C 180,E1 -13988.386,E2 -13988.386} C_VEL
LIN {X 0,Y 340.697,Z 146.046,A -85,B 0,C 180,E1 -13992.045,E2 -13992.045} C_VEL
LIN {X 0,Y 340.65,Z 146.055,A -85,B 0,C 180,E1 -13996.227,E2 -13996.227} C_VEL
LIN {X 0,Y 340.687,Z 146.047,A -85,B 0,C 180,E1 -13999.753,E2 -13999.753} C_VEL
LIN {X 0,Y 340.704,Z 146.043,A -85,B 0,C 180,E1 -14003.259,E2 -14003.259} C_VEL
LIN {X 0,Y 340.692,Z 146.048,A -85,B 0,C 180,E1 -14006.154,E2 -14006.154} C_VEL
LIN {X 0,Y 340.773,Z 146.035,A -85,B 0,C 180,E1 -14010.333,E2 -14010.333} C_VEL
LIN {X 0,Y 340.803,Z 146.03,A -85,B 0,C 180,E1 -14013.02,E2 -14013.02} C_VEL
LIN {X 0,Y 340.752,Z 146.041,A -85,B 0,C 180,E1 -14015.638,E2 -14015.638} C_VEL
LIN {X 0,Y 340.736,Z 146.043,A -85,B 0,C 180,E1 -14019.474,E2 -14019.474} C_VEL
LIN {X 0,Y 340.857,Z 146.025,A -85,B 0,C 180,E1 -14021.984,E2 -14021.984} C_VEL
LIN {X 0,Y 340.868,Z 146.025,A -85,B 0,C 180,E1 -14025.705,E2 -14025.705} C_VEL
LIN {X 0,Y 340.869,Z 146.027,A -85,B 0,C 180,E1 -14029.306,E2 -14029.306} C_VEL
LIN {X 0,Y 341.074,Z 145.998,A -85,B 0,C 180,E1 -14032.898,E2 -14032.898} C_VEL
LIN {X 0,Y 341.168,Z 145.986,A -85,B 0,C 180,E1 -14037.639,E2 -14037.639} C_VEL
LIN {X 0,Y 341.295,Z 145.969,A -85,B 0,C 180,E1 -14040,E2 -14040} C_VEL
LIN {X 0,Y 341.168,Z 145.985,A -85,B 0,C 180,E1 -14042.361,E2 -14042.361} C_VEL
LIN {X 0,Y 341.059,Z 146.002,A -85,B 0,C 180,E1 -14047.102,E2 -14047.102} C_VEL
LIN {X 0,Y 340.87,Z 146.026,A -85,B 0,C 180,E1 -14050.694,E2 -14050.694} C_VEL
LIN {X 0,Y 340.862,Z 146.025,A -85,B 0,C 180,E1 -14054.325,E2 -14054.325} C_VEL
LIN {X 0,Y 340.837,Z 146.03,A -85,B 0,C 180,E1 -14058.467,E2 -14058.467} C_VEL
LIN {X 0,Y 340.717,Z 146.041,A -85,B 0,C 180,E1 -14061.842,E2 -14061.842} C_VEL
LIN {X 0,Y 340.772,Z 146.034,A -85,B 0,C 180,E1 -14065.665,E2 -14065.665} C_VEL
LIN {X 0,Y 340.741,Z 146.043,A -85,B 0,C 180,E1 -14068.32,E2 -14068.32} C_VEL
LIN {X 0,Y 340.703,Z 146.043,A -85,B 0,C 180,E1 -14071.044,E2 -14071.044} C_VEL
LIN {X 0,Y 340.718,Z 146.04,A -85,B 0,C 180,E1 -14075.279,E2 -14075.279} C_VEL
LIN {X 0,Y 340.718,Z 146.044,A -85,B 0,C 180,E1 -14078.388,E2 -14078.388} C_VEL
LIN {X 0,Y 340.73,Z 146.045,A -85,B 0,C 180,E1 -14082.052,E2 -14082.052} C_VEL
LIN {X 0,Y 340.664,Z 146.05,A -85,B 0,C 180,E1 -14086.225,E2 -14086.225} C_VEL
LIN {X 0,Y 340.705,Z 146.042,A -85,B 0,C 180,E1 -14088.694,E2 -14088.694} C_VEL
LIN {X 0,Y 340.74,Z 146.043,A -85,B 0,C 180,E1 -14091.774,E2 -14091.774} C_VEL
LIN {X 0,Y 340.724,Z 146.044,A -85,B 0,C 180,E1 -14095.596,E2 -14095.596} C_VEL
LIN {X 0,Y 340.74,Z 146.156,A -85,B 0,C 180,E1 -14098.311,E2 -14098.311} C_VEL
LIN {X 0,Y 343.88,Z 160.415,A -85,B 0,C 180,E1 -14101.962,E2 -14101.962} C_VEL
LIN {X 0,Y 344.947,Z 167.538,A -85,B 0,C 180,E1 -14103.698,E2 -14103.698} C_VEL
LIN {X 0,Y 343.369,Z 182.868,A -85,B 0,C 180,E1 -14107.144,E2 -14107.144} C_VEL
LIN {X 0,Y 347.986,Z 215.819,A -85,B 0,C 180,E1 -14108.186,E2 -14108.186} C_VEL
LIN {X 0,Y 348.813,Z 224.034,A -85,B 0,C 180,E1 -14108.422,E2 -14108.422} C_VEL
LIN {X 0,Y 347.458,Z 291.927,A -85,B 0,C 180,E1 -14109.927,E2 -14109.927} C_VEL
LIN {X 0,Y 346.723,Z 305.644,A -85,B 0,C 180,E1 -14110.461,E2 -14110.461} C_VEL
LIN {X 0,Y 345.769,Z 318.081,A -85,B 0,C 180,E1 -14111.176,E2 -14111.176} C_VEL
LIN {X 0,Y 344.74,Z 329.235,A -85,B 0,C 180,E1 -14112.041,E2 -14112.041} C_VEL
LIN {X 0,Y 343.568,Z 340.874,A -85,B 0,C 180,E1 -14113.206,E2 -14113.206} C_VEL
LIN {X 0,Y 342.481,Z 351.377,A -85,B 0,C 180,E1 -14114.528,E2 -14114.528} C_VEL
LIN {X 0,Y 341.524,Z 360.824,A -85,B 0,C 180,E1 -14116.008,E2 -14116.008} C_VEL
LIN {X 0,Y 340.53,Z 369.949,A -85,B 0,C 180,E1 -14117.787,E2 -14117.787} C_VEL
LIN {X 0,Y 339.845,Z 377.298,A -85,B 0,C 180,E1 -14119.575,E2 -14119.575} C_VEL
LIN {X 0,Y 339.489,Z 382.253,A -85,B 0,C 180,E1 -14121.068,E2 -14121.068} C_VEL
LIN {X 0,Y 339.247,Z 387.054,A -85,B 0,C 180,E1 -14122.86,E2 -14122.86} C_VEL
LIN {X 0,Y 339.111,Z 390.52,A -85,B 0,C 180,E1 -14124.549,E2 -14124.549} C_VEL
LIN {X 0,Y 339.147,Z 393.305,A -85,B 0,C 180,E1 -14126.436,E2 -14126.436} C_VEL
LIN {X 0,Y 339.181,Z 394.516,A -85,B 0,C 180,E1 -14127.625,E2 -14127.625} C_VEL
LIN {X 0,Y 339.303,Z 395.278,A -85,B 0,C 180,E1 -14128.813,E2 -14128.813} C_VEL
LIN {X 0,Y 339.33,Z 395.616,A -85,B 0,C 180,E1 -14130,E2 -14130} C_VEL
LIN {X 0,Y 339.258,Z 395.551,A -85,B 0,C 180,E1 -14131.187,E2 -14131.187} C_VEL
LIN {X 0,Y 339.137,Z 395.086,A -85,B 0,C 180,E1 -14132.375,E2 -14132.375} C_VEL
LIN {X 0,Y 339.126,Z 394.186,A -85,B 0,C 180,E1 -14133.564,E2 -14133.564} C_VEL
LIN {X 0,Y 339.116,Z 391.275,A -85,B 0,C 180,E1 -14135.857,E2 -14135.857} C_VEL
LIN {X 0,Y 339.324,Z 387.679,A -85,B 0,C 180,E1 -14137.737,E2 -14137.737} C_VEL
LIN {X 0,Y 339.662,Z 383.142,A -85,B 0,C 180,E1 -14139.528,E2 -14139.528} C_VEL
LIN {X 0,Y 340.216,Z 377.402,A -85,B 0,C 180,E1 -14141.317,E2 -14141.317} C_VEL
LIN {X 0,Y 341.206,Z 370.282,A -85,B 0,C 180,E1 -14143.095,E2 -14143.095} C_VEL
LIN {X 0,Y 342.337,Z 361.68,A -85,B 0,C 180,E1 -14144.817,E2 -14144.817} C_VEL
LIN {X 0,Y 343.511,Z 352.337,A -85,B 0,C 180,E1 -14146.338,E2 -14146.338} C_VEL
LIN {X 0,Y 344.815,Z 342.411,A -85,B 0,C 180,E1 -14147.649,E2 -14147.649} C_VEL
LIN {X 0,Y 346.291,Z 331.497,A -85,B 0,C 180,E1 -14148.795,E2 -14148.795} C_VEL
LIN {X 0,Y 347.632,Z 319.334,A -85,B 0,C 180,E1 -14149.793,E2 -14149.793} C_VEL
LIN {X 0,Y 348.846,Z 306.706,A -85,B 0,C 180,E1 -14150.567,E2 -14150.567} C_VEL
LIN {X 0,Y 349.748,Z 293.311,A -85,B 0,C 180,E1 -14151.127,E2 -14151.127} C_VEL
LIN {X 0,Y 350.282,Z 275.673,A -85,B 0,C 180,E1 -14151.569,E2 -14151.569} C_VEL
LIN {X 0,Y 351.459,Z 222.227,A -85,B 0,C 180,E1 -14152.759,E2 -14152.759} C_VEL
LIN {X 0,Y 348.198,Z 199.284,A -85,B 0,C 180,E1 -14153.585,E2 -14153.585} C_VEL
LIN {X 0,Y 344.689,Z 180.661,A -85,B 0,C 180,E1 -14154.354,E2 -14154.354} C_VEL
LIN {X 0,Y 345.932,Z 169.556,A -85,B 0,C 180,E1 -14156.873,E2 -14156.873} C_VEL
LIN {X 0,Y 344.112,Z 159.979,A -85,B 0,C 180,E1 -14159.351,E2 -14159.351} C_VEL
LIN {X 0,Y 341.13,Z 147.726,A -85,B 0,C 180,E1 -14162.738,E2 -14162.738} C_VEL
LIN {X 0,Y 340.694,Z 146.05,A -85,B 0,C 180,E1 -14163.225,E2 -14163.225} C_VEL
LIN {X 0,Y 340.707,Z 146.049,A -85,B 0,C 180,E1 -14166.741,E2 -14166.741} C_VEL
LIN {X 0,Y 340.71,Z 146.052,A -85,B 0,C 180,E1 -14170.251,E2 -14170.251} C_VEL
LIN {X 0,Y 340.702,Z 146.048,A -85,B 0,C 180,E1 -14172.9,E2 -14172.9} C_VEL
LIN {X 0,Y 340.711,Z 146.047,A -85,B 0,C 180,E1 -14177.101,E2 -14177.101} C_VEL
LIN {X 0,Y 340.71,Z 146.044,A -85,B 0,C 180,E1 -14180.249,E2 -14180.249} C_VEL
LIN {X 0,Y 340.71,Z 146.043,A -85,B 0,C 180,E1 -14183.559,E2 -14183.559} C_VEL
LIN {X 0,Y 340.691,Z 146.045,A -85,B 0,C 180,E1 -14186.153,E2 -14186.153} C_VEL
LIN {X 0,Y 340.774,Z 146.03,A -85,B 0,C 180,E1 -14190.332,E2 -14190.332} C_VEL
LIN {X 0,Y 340.804,Z 146.031,A -85,B 0,C 180,E1 -14193.02,E2 -14193.02} C_VEL
LIN {X 0,Y 340.753,Z 146.04,A -85,B 0,C 180,E1 -14195.638,E2 -14195.638} C_VEL
LIN {X 0,Y 340.737,Z 146.041,A -85,B 0,C 180,E1 -14199.473,E2 -14199.473} C_VEL
LIN {X 0,Y 340.857,Z 146.023,A -85,B 0,C 180,E1 -14201.984,E2 -14201.984} C_VEL
LIN {X 0,Y 340.868,Z 146.021,A -85,B 0,C 180,E1 -14205.705,E2 -14205.705} C_VEL
LIN {X 0,Y 340.869,Z 146.02,A -85,B 0,C 180,E1 -14209.306,E2 -14209.306} C_VEL
LIN {X 0,Y 341.074,Z 145.993,A -85,B 0,C 180,E1 -14212.898,E2 -14212.898} C_VEL
LIN {X 0,Y 341.168,Z 145.988,A -85,B 0,C 180,E1 -14217.639,E2 -14217.639} C_VEL
LIN {X 0,Y 341.295,Z 145.966,A -85,B 0,C 180,E1 -14220,E2 -14220} C_VEL
LIN {X 0,Y 341.168,Z 145.987,A -85,B 0,C 180,E1 -14222.361,E2 -14222.361} C_VEL
LIN {X 0,Y 341.056,Z 146.003,A -85,B 0,C 180,E1 -14227.102,E2 -14227.102} C_VEL
LIN {X 0,Y 340.869,Z 146.027,A -85,B 0,C 180,E1 -14230.694,E2 -14230.694} C_VEL
LIN {X 0,Y 340.861,Z 146.025,A -85,B 0,C 180,E1 -14234.325,E2 -14234.325} C_VEL
LIN {X 0,Y 340.836,Z 146.029,A -85,B 0,C 180,E1 -14238.467,E2 -14238.467} C_VEL
LIN {X 0,Y 340.752,Z 146.041,A -85,B 0,C 180,E1 -14241.857,E2 -14241.857} C_VEL
LIN {X 0,Y 340.77,Z 146.04,A -85,B 0,C 180,E1 -14245.664,E2 -14245.664} C_VEL
LIN {X 0,Y 340.821,Z 146.111,A -85,B 0,C 180,E1 -14247.36,E2 -14247.36} C_VEL
LIN {X 0,Y 341.665,Z 149.612,A -85,B 0,C 180,E1 -14248.445,E2 -14248.445} C_VEL
LIN {X 0,Y 350.001,Z 168.417,A -85,B 0,C 180,E1 -14249.657,E2 -14249.657} C_VEL
LIN {X 0,Y 352.706,Z 175.716,A -85,B 0,C 180,E1 -14250.063,E2 -14250.063} C_VEL
LIN {X 0,Y 350.483,Z 257.297,A -85,B 0,C 180,E1 -14251.901,E2 -14251.901} C_VEL
LIN {X 0,Y 349.856,Z 270.179,A -85,B 0,C 180,E1 -14252.423,E2 -14252.423} C_VEL
LIN {X 0,Y 349.083,Z 282.906,A -85,B 0,C 180,E1 -14253.186,E2 -14253.186} C_VEL
LIN {X 0,Y 348.04,Z 294.459,A -85,B 0,C 180,E1 -14254.115,E2 -14254.115} C_VEL
LIN {X 0,Y 346.831,Z 305.707,A -85,B 0,C 180,E1 -14255.275,E2 -14255.275} C_VEL
LIN {X 0,Y 345.613,Z 315.683,A -85,B 0,C 180,E1 -14256.561,E2 -14256.561} C_VEL
LIN {X 0,Y 344.399,Z 324.475,A -85,B 0,C 180,E1 -14257.957,E2 -14257.957} C_VEL
LIN {X 0,Y 343.274,Z 331.943,A -85,B 0,C 180,E1 -14259.396,E2 -14259.396} C_VEL
LIN {X 0,Y 342.135,Z 339.139,A -85,B 0,C 180,E1 -14261.096,E2 -14261.096} C_VEL
LIN {X 0,Y 341.286,Z 344.956,A -85,B 0,C 180,E1 -14262.809,E2 -14262.809} C_VEL
LIN {X 0,Y 340.556,Z 349.684,A -85,B 0,C 180,E1 -14264.559,E2 -14264.559} C_VEL
LIN {X 0,Y 340.015,Z 353.371,A -85,B 0,C 180,E1 -14266.339,E2 -14266.339} C_VEL
LIN {X 0,Y 339.498,Z 356.517,A -85,B 0,C 180,E1 -14268.514,E2 -14268.514} C_VEL
LIN {X 0,Y 339.24,Z 357.869,A -85,B 0,C 180,E1 -14270.043,E2 -14270.043} C_VEL
LIN {X 0,Y 339.105,Z 358.622,A -85,B 0,C 180,E1 -14271.957,E2 -14271.957} C_VEL
LIN {X 0,Y 339.074,Z 358.31,A -85,B 0,C 180,E1 -14273.935,E2 -14273.935} C_VEL
LIN {X 0,Y 339.2,Z 356.815,A -85,B 0,C 180,E1 -14275.985,E2 -14275.985} C_VEL
LIN {X 0,Y 339.514,Z 354.036,A -85,B 0,C 180,E1 -14278.071,E2 -14278.071} C_VEL
LIN {X 0,Y 340.002,Z 349.604,A -85,B 0,C 180,E1 -14280.259,E2 -14280.259} C_VEL
LIN {X 0,Y 340.507,Z 344.458,A -85,B 0,C 180,E1 -14282.139,E2 -14282.139} C_VEL
LIN {X 0,Y 341.241,Z 337.776,A -85,B 0,C 180,E1 -14284.046,E2 -14284.046} C_VEL
LIN {X 0,Y 342.075,Z 330.328,A -85,B 0,C 180,E1 -14285.739,E2 -14285.739} C_VEL
LIN {X 0,Y 343.013,Z 322.307,A -85,B 0,C 180,E1 -14287.221,E2 -14287.221} C_VEL
LIN {X 0,Y 344.045,Z 312.206,A -85,B 0,C 180,E1 -14288.741,E2 -14288.741} C_VEL
LIN {X 0,Y 345.106,Z 301.322,A -85,B 0,C 180,E1 -14290.056,E2 -14290.056} C_VEL
LIN {X 0,Y 346.108,Z 289.258,A -85,B 0,C 180,E1 -14291.192,E2 -14291.192} C_VEL
LIN {X 0,Y 346.871,Z 276.979,A -85,B 0,C 180,E1 -14292.082,E2 -14292.082} C_VEL
LIN {X 0,Y 347.542,Z 263.885,A -85,B 0,C 180,E1 -14292.76,E2 -14292.76} C_VEL
LIN {X 0,Y 347.967,Z 250.646,A -85,B 0,C 180,E1 -14293.198,E2 -14293.198} C_VEL
LIN {X 0,Y 349.576,Z 172.339,A -85,B 0,C 180,E1 -14294.906,E2 -14294.906} C_VEL
LIN {X 0,Y 346.339,Z 161.896,A -85,B 0,C 180,E1 -14295.341,E2 -14295.341} C_VEL
LIN {X 0,Y 341.209,Z 147.549,A -85,B 0,C 180,E1 -14296.006,E2 -14296.006} C_VEL
LIN {X 0,Y 340.884,Z 146.024,A -85,B 0,C 180,E1 -14296.455,E2 -14296.455} C_VEL
LIN {X 0,Y 340.913,Z 146.016,A -85,B 0,C 180,E1 -14300.507,E2 -14300.507} C_VEL
LIN {X 0,Y 341.058,Z 145.999,A -85,B 0,C 180,E1 -14302.898,E2 -14302.898} C_VEL
LIN {X 0,Y 341.167,Z 145.988,A -85,B 0,C 180,E1 -14307.639,E2 -14307.639} C_VEL
LIN {X 0,Y 341.295,Z 145.969,A -85,B 0,C 180,E1 -14310,E2 -14310} C_VEL
LIN {X 0,Y 341.168,Z 145.984,A -85,B 0,C 180,E1 -14312.361,E2 -14312.361} C_VEL
LIN {X 0,Y 341.009,Z 146.01,A -85,B 0,C 180,E1 -14317.103,E2 -14317.103} C_VEL
LIN {X 0,Y 340.848,Z 146.027,A -85,B 0,C 180,E1 -14320.694,E2 -14320.694} C_VEL
LIN {X 0,Y 340.863,Z 146.023,A -85,B 0,C 180,E1 -14324.325,E2 -14324.325} C_VEL
LIN {X 0,Y 340.785,Z 146.034,A -85,B 0,C 180,E1 -14328.44,E2 -14328.44} C_VEL
LIN {X 0,Y 340.717,Z 146.041,A -85,B 0,C 180,E1 -14331.842,E2 -14331.842} C_VEL
LIN {X 0,Y 340.72,Z 146.04,A -85,B 0,C 180,E1 -14333.846,E2 -14333.846} C_VEL
LIN {X 0,Y 340.096,Z 146.123,A -85,B 0,C 180,E1 -14334.832,E2 -14334.832} C_VEL
LIN {X 0,Y 337.288,Z 146.475,A -85,B 0,C 180,E1 -14336.438,E2 -14336.438} C_VEL
LIN {X 0,Y 334.869,Z 146.777,A -85,B 0,C 180,E1 -14337.737,E2 -14337.737} C_VEL
LIN {X 0,Y 333.803,Z 146.907,A -85,B 0,C 180,E1 -14338.743,E2 -14338.743} C_VEL
LIN {X 0,Y 333.702,Z 146.916,A -85,B 0,C 180,E1 -14339.084,E2 -14339.084} C_VEL
LIN {X 0,Y 333.635,Z 146.923,A -85,B 0,C 180,E1 -14343.208,E2 -14343.208} C_VEL
LIN {X 0,Y 333.675,Z 146.921,A -85,B 0,C 180,E1 -14346.139,E2 -14346.139} C_VEL
LIN {X 0,Y 333.645,Z 146.922,A -85,B 0,C 180,E1 -14349.192,E2 -14349.192} C_VEL
LIN {X 0,Y 333.631,Z 146.927,A -85,B 0,C 180,E1 -14352.5,E2 -14352.5} C_VEL
LIN {X 0,Y 333.595,Z 146.931,A -85,B 0,C 180,E1 -14355.955,E2 -14355.955} C_VEL
LIN {X 0,Y 333.646,Z 146.922,A -85,B 0,C 180,E1 -14359.315,E2 -14359.315} C_VEL
LIN {X 0,Y 333.664,Z 146.919,A -85,B 0,C 180,E1 -14363.168,E2 -14363.168} C_VEL
LIN {X 0,Y 333.637,Z 146.923,A -85,B 0,C 180,E1 -14366.792,E2 -14366.792} C_VEL
LIN {X 0,Y 333.701,Z 146.919,A -85,B 0,C 180,E1 -14369.71,E2 -14369.71} C_VEL
LIN {X 0,Y 333.742,Z 146.91,A -85,B 0,C 180,E1 -14372.401,E2 -14372.401} C_VEL
LIN {X 0,Y 333.724,Z 146.913,A -85,B 0,C 180,E1 -14375.091,E2 -14375.091} C_VEL
LIN {X 0,Y 333.674,Z 146.919,A -85,B 0,C 180,E1 -14379.019,E2 -14379.019} C_VEL
LIN {X 0,Y 333.793,Z 146.908,A -85,B 0,C 180,E1 -14381.59,E2 -14381.59} C_VEL
LIN {X 0,Y 333.807,Z 146.906,A -85,B 0,C 180,E1 -14385.577,E2 -14385.577} C_VEL
LIN {X 0,Y 333.832,Z 146.901,A -85,B 0,C 180,E1 -14389.078,E2 -14389.078} C_VEL
LIN {X 0,Y 334.024,Z 146.875,A -85,B 0,C 180,E1 -14392.748,E2 -14392.748} C_VEL
LIN {X 0,Y 333.81,Z 146.906,A -85,B 0,C 180,E1 -14395.169,E2 -14395.169} C_VEL
LIN {X 0,Y 334.105,Z 146.866,A -85,B 0,C 180,E1 -14397.589,E2 -14397.589} C_VEL
LIN {X 0,Y 334.246,Z 146.847,A -85,B 0,C 180,E1 -14400,E2 -14400} C_VEL
LIN {X 0,Y 334.106,Z 146.865,A -85,B 0,C 180,E1 -14402.411,E2 -14402.411} C_VEL
LIN {X 0,Y 334.013,Z 146.876,A -85,B 0,C 180,E1 -14406.039,E2 -14406.039} C_VEL
LIN {X 0,Y 333.984,Z 146.882,A -85,B 0,C 180,E1 -14408.502,E2 -14408.502} C_VEL
LIN {X 0,Y 333.79,Z 146.904,A -85,B 0,C 180,E1 -14412.155,E2 -14412.155} C_VEL
LIN {X 0,Y 333.777,Z 146.905,A -85,B 0,C 180,E1 -14415.886,E2 -14415.886} C_VEL
LIN {X 0,Y 333.796,Z 146.908,A -85,B 0,C 180,E1 -14418.656,E2 -14418.656} C_VEL
LIN {X 0,Y 333.656,Z 146.923,A -85,B 0,C 180,E1 -14422.281,E2 -14422.281} C_VEL
LIN {X 0,Y 333.735,Z 146.914,A -85,B 0,C 180,E1 -14426.247,E2 -14426.247} C_VEL
LIN {X 0,Y 333.711,Z 146.914,A -85,B 0,C 180,E1 -14428.972,E2 -14428.972} C_VEL
LIN {X 0,Y 333.643,Z 146.925,A -85,B 0,C 180,E1 -14432.587,E2 -14432.587} C_VEL
LIN {X 0,Y 333.677,Z 146.923,A -85,B 0,C 180,E1 -14436.139,E2 -14436.139} C_VEL
LIN {X 0,Y 333.673,Z 146.918,A -85,B 0,C 180,E1 -14439.189,E2 -14439.189} C_VEL
LIN {X 0,Y 333.661,Z 146.921,A -85,B 0,C 180,E1 -14442.506,E2 -14442.506} C_VEL
LIN {X 0,Y 333.612,Z 146.932,A -85,B 0,C 180,E1 -14445.958,E2 -14445.958} C_VEL
LIN {X 0,Y 333.657,Z 146.921,A -85,B 0,C 180,E1 -14449.314,E2 -14449.314} C_VEL
LIN {X 0,Y 333.657,Z 146.921,A -85,B 0,C 180,E1 -14452.35,E2 -14452.35} C_VEL
LIN {X 0,Y 333.676,Z 146.92,A -85,B 0,C 180,E1 -14455.342,E2 -14455.342} C_VEL
LIN {X 0,Y 333.674,Z 146.939,A -85,B 0,C 180,E1 -14457.947,E2 -14457.947} C_VEL
LIN {X 0,Y 336.893,Z 161.531,A -85,B 0,C 180,E1 -14461.768,E2 -14461.768} C_VEL
LIN {X 0,Y 337.981,Z 168.065,A -85,B 0,C 180,E1 -14463.399,E2 -14463.399} C_VEL
LIN {X 0,Y 336.547,Z 182.086,A -85,B 0,C 180,E1 -14466.624,E2 -14466.624} C_VEL
LIN {X 0,Y 336.512,Z 182.523,A -85,B 0,C 180,E1 -14466.724,E2 -14466.724} C_VEL
LIN {X 0,Y 341.616,Z 219.324,A -85,B 0,C 180,E1 -14467.908,E2 -14467.908} C_VEL
LIN {X 0,Y 342.08,Z 225.53,A -85,B 0,C 180,E1 -14468.081,E2 -14468.081} C_VEL
LIN {X 0,Y 340.683,Z 291.981,A -85,B 0,C 180,E1 -14469.588,E2 -14469.588} C_VEL
LIN {X 0,Y 339.9,Z 305.544,A -85,B 0,C 180,E1 -14470.131,E2 -14470.131} C_VEL
LIN {X 0,Y 338.938,Z 317.902,A -85,B 0,C 180,E1 -14470.86,E2 -14470.86} C_VEL
LIN {X 0,Y 337.794,Z 329.797,A -85,B 0,C 180,E1 -14471.815,E2 -14471.815} C_VEL
LIN {X 0,Y 336.589,Z 341.265,A -85,B 0,C 180,E1 -14473.003,E2 -14473.003} C_VEL
LIN {X 0,Y 335.408,Z 352.168,A -85,B 0,C 180,E1 -14474.433,E2 -14474.433} C_VEL
LIN {X 0,Y 334.385,Z 361.758,A -85,B 0,C 180,E1 -14476.013,E2 -14476.013} C_VEL
LIN {X 0,Y 333.399,Z 370.665,A -85,B 0,C 180,E1 -14477.831,E2 -14477.831} C_VEL
LIN {X 0,Y 332.731,Z 377.768,A -85,B 0,C 180,E1 -14479.657,E2 -14479.657} C_VEL
LIN {X 0,Y 332.332,Z 383.439,A -85,B 0,C 180,E1 -14481.487,E2 -14481.487} C_VEL
LIN {X 0,Y 332.112,Z 387.876,A -85,B 0,C 180,E1 -14483.316,E2 -14483.316} C_VEL
LIN {X 0,Y 332.069,Z 391.206,A -85,B 0,C 180,E1 -14485.144,E2 -14485.144} C_VEL
LIN {X 0,Y 332.069,Z 392.848,A -85,B 0,C 180,E1 -14486.36,E2 -14486.36} C_VEL
LIN {X 0,Y 332.086,Z 394.074,A -85,B 0,C 180,E1 -14487.574,E2 -14487.574} C_VEL
LIN {X 0,Y 332.207,Z 394.865,A -85,B 0,C 180,E1 -14488.788,E2 -14488.788} C_VEL
LIN {X 0,Y 332.251,Z 395.219,A -85,B 0,C 180,E1 -14490,E2 -14490} C_VEL
LIN {X 0,Y 332.162,Z 395.165,A -85,B 0,C 180,E1 -14491.212,E2 -14491.212} C_VEL
LIN {X 0,Y 332.045,Z 394.715,A -85,B 0,C 180,E1 -14492.426,E2 -14492.426} C_VEL
LIN {X 0,Y 332.048,Z 393.842,A -85,B 0,C 180,E1 -14493.64,E2 -14493.64} C_VEL
LIN {X 0,Y 332.018,Z 391.234,A -85,B 0,C 180,E1 -14495.801,E2 -14495.801} C_VEL
LIN {X 0,Y 332.244,Z 387.394,A -85,B 0,C 180,E1 -14497.903,E2 -14497.903} C_VEL
LIN {X 0,Y 332.624,Z 382.897,A -85,B 0,C 180,E1 -14499.731,E2 -14499.731} C_VEL
LIN {X 0,Y 333.234,Z 377.205,A -85,B 0,C 180,E1 -14501.558,E2 -14501.558} C_VEL
LIN {X 0,Y 334.282,Z 370.137,A -85,B 0,C 180,E1 -14503.371,E2 -14503.371} C_VEL
LIN {X 0,Y 335.414,Z 361.941,A -85,B 0,C 180,E1 -14505.066,E2 -14505.066} C_VEL
LIN {X 0,Y 336.691,Z 352.312,A -85,B 0,C 180,E1 -14506.679,E2 -14506.679} C_VEL
LIN {X 0,Y 338.241,Z 341.26,A -85,B 0,C 180,E1 -14508.16,E2 -14508.16} C_VEL
LIN {X 0,Y 339.76,Z 330.122,A -85,B 0,C 180,E1 -14509.327,E2 -14509.327} C_VEL
LIN {X 0,Y 341.18,Z 317.718,A -85,B 0,C 180,E1 -14510.341,E2 -14510.341} C_VEL
LIN {X 0,Y 342.342,Z 306.03,A -85,B 0,C 180,E1 -14511.055,E2 -14511.055} C_VEL
LIN {X 0,Y 343.299,Z 292.535,A -85,B 0,C 180,E1 -14511.623,E2 -14511.623} C_VEL
LIN {X 0,Y 343.939,Z 272.286,A -85,B 0,C 180,E1 -14512.129,E2 -14512.129} C_VEL
LIN {X 0,Y 345.078,Z 223.112,A -85,B 0,C 180,E1 -14513.25,E2 -14513.25} C_VEL
LIN {X 0,Y 341.944,Z 200.794,A -85,B 0,C 180,E1 -14514.076,E2 -14514.076} C_VEL
LIN {X 0,Y 338.049,Z 180.212,A -85,B 0,C 180,E1 -14514.957,E2 -14514.957} C_VEL
LIN {X 0,Y 339.059,Z 170.896,A -85,B 0,C 180,E1 -14517.13,E2 -14517.13} C_VEL
LIN {X 0,Y 337.146,Z 161.11,A -85,B 0,C 180,E1 -14519.733,E2 -14519.733} C_VEL
LIN {X 0,Y 334.527,Z 150.23,A -85,B 0,C 180,E1 -14522.822,E2 -14522.822} C_VEL
LIN {X 0,Y 333.668,Z 146.926,A -85,B 0,C 180,E1 -14523.838,E2 -14523.838} C_VEL
LIN {X 0,Y 333.657,Z 146.929,A -85,B 0,C 180,E1 -14527.65,E2 -14527.65} C_VEL
LIN {X 0,Y 333.656,Z 146.926,A -85,B 0,C 180,E1 -14530.766,E2 -14530.766} C_VEL
LIN {X 0,Y 333.611,Z 146.935,A -85,B 0,C 180,E1 -14534.253,E2 -14534.253} C_VEL
LIN {X 0,Y 333.674,Z 146.924,A -85,B 0,C 180,E1 -14537.623,E2 -14537.623} C_VEL
LIN {X 0,Y 333.677,Z 146.916,A -85,B 0,C 180,E1 -14541.196,E2 -14541.196} C_VEL
LIN {X 0,Y 333.685,Z 146.919,A -85,B 0,C 180,E1 -14545.225,E2 -14545.225} C_VEL
LIN {X 0,Y 333.697,Z 146.916,A -85,B 0,C 180,E1 -14549.637,E2 -14549.637} C_VEL
LIN {X 0,Y 333.742,Z 146.91,A -85,B 0,C 180,E1 -14552.401,E2 -14552.401} C_VEL
LIN {X 0,Y 333.725,Z 146.91,A -85,B 0,C 180,E1 -14555.09,E2 -14555.09} C_VEL
LIN {X 0,Y 333.674,Z 146.917,A -85,B 0,C 180,E1 -14559.018,E2 -14559.018} C_VEL
LIN {X 0,Y 333.793,Z 146.899,A -85,B 0,C 180,E1 -14561.589,E2 -14561.589} C_VEL
LIN {X 0,Y 333.807,Z 146.899,A -85,B 0,C 180,E1 -14565.576,E2 -14565.576} C_VEL
LIN {X 0,Y 333.832,Z 146.895,A -85,B 0,C 180,E1 -14569.078,E2 -14569.078} C_VEL
LIN {X 0,Y 334.024,Z 146.87,A -85,B 0,C 180,E1 -14572.747,E2 -14572.747} C_VEL
LIN {X 0,Y 333.809,Z 146.902,A -85,B 0,C 180,E1 -14575.169,E2 -14575.169} C_VEL
LIN {X 0,Y 334.105,Z 146.868,A -85,B 0,C 180,E1 -14577.589,E2 -14577.589} C_VEL
LIN {X 0,Y 334.246,Z 146.844,A -85,B 0,C 180,E1 -14580,E2 -14580} C_VEL
LIN {X 0,Y 334.105,Z 146.866,A -85,B 0,C 180,E1 -14582.411,E2 -14582.411} C_VEL
LIN {X 0,Y 333.99,Z 146.878,A -85,B 0,C 180,E1 -14586.597,E2 -14586.597} C_VEL
LIN {X 0,Y 333.849,Z 146.9,A -85,B 0,C 180,E1 -14589.695,E2 -14589.695} C_VEL
LIN {X 0,Y 333.795,Z 146.905,A -85,B 0,C 180,E1 -14593.391,E2 -14593.391} C_VEL
LIN {X 0,Y 333.745,Z 146.914,A -85,B 0,C 180,E1 -14597.146,E2 -14597.146} C_VEL
LIN {X 0,Y 333.737,Z 146.913,A -85,B 0,C 180,E1 -14599.69,E2 -14599.69} C_VEL
LIN {X 0,Y 333.69,Z 146.924,A -85,B 0,C 180,E1 -14602.278,E2 -14602.278} C_VEL
LIN {X 0,Y 333.731,Z 146.915,A -85,B 0,C 180,E1 -14606.246,E2 -14606.246} C_VEL
LIN {X 0,Y 333.782,Z 147.141,A -85,B 0,C 180,E1 -14606.832,E2 -14606.832} C_VEL
LIN {X 0,Y 334.578,Z 150.213,A -85,B 0,C 180,E1 -14607.781,E2 -14607.781} C_VEL
LIN {X 0,Y 342.908,Z 168.48,A -85,B 0,C 180,E1 -14609.044,E2 -14609.044} C_VEL
LIN {X 0,Y 346.334,Z 176.973,A -85,B 0,C 180,E1 -14609.557,E2 -14609.557} C_VEL
LIN {X 0,Y 344.073,Z 257.426,A -85,B 0,C 180,E1 -14611.407,E2 -14611.407} C_VEL
LIN {X 0,Y 343.4,Z 270.63,A -85,B 0,C 180,E1 -14611.951,E2 -14611.951} C_VEL
LIN {X 0,Y 342.621,Z 282.416,A -85,B 0,C 180,E1 -14612.662,E2 -14612.662} C_VEL
LIN {X 0,Y 341.551,Z 294.271,A -85,B 0,C 180,E1 -14613.619,E2 -14613.619} C_VEL
LIN {X 0,Y 340.232,Z 305.912,A -85,B 0,C 180,E1 -14614.834,E2 -14614.834} C_VEL
LIN {X 0,Y 338.862,Z 316.466,A -85,B 0,C 180,E1 -14616.221,E2 -14616.221} C_VEL
LIN {X 0,Y 337.536,Z 325.498,A -85,B 0,C 180,E1 -14617.701,E2 -14617.701} C_VEL
LIN {X 0,Y 336.235,Z 333.642,A -85,B 0,C 180,E1 -14619.343,E2 -14619.343} C_VEL
LIN {X 0,Y 335.143,Z 340.256,A -85,B 0,C 180,E1 -14620.982,E2 -14620.982} C_VEL
LIN {X 0,Y 334.157,Z 346.747,A -85,B 0,C 180,E1 -14623.006,E2 -14623.006} C_VEL
LIN {X 0,Y 333.327,Z 351.737,A -85,B 0,C 180,E1 -14625.065,E2 -14625.065} C_VEL
LIN {X 0,Y 332.854,Z 354.685,A -85,B 0,C 180,E1 -14626.669,E2 -14626.669} C_VEL
LIN {X 0,Y 332.581,Z 356.152,A -85,B 0,C 180,E1 -14627.698,E2 -14627.698} C_VEL
LIN {X 0,Y 332.21,Z 358.07,A -85,B 0,C 180,E1 -14629.604,E2 -14629.604} C_VEL
LIN {X 0,Y 332.043,Z 358.986,A -85,B 0,C 180,E1 -14631.548,E2 -14631.548} C_VEL
LIN {X 0,Y 331.985,Z 358.811,A -85,B 0,C 180,E1 -14633.648,E2 -14633.648} C_VEL
LIN {X 0,Y 332.075,Z 357.555,A -85,B 0,C 180,E1 -14635.628,E2 -14635.628} C_VEL
LIN {X 0,Y 332.398,Z 354.984,A -85,B 0,C 180,E1 -14637.75,E2 -14637.75} C_VEL
LIN {X 0,Y 332.84,Z 350.896,A -85,B 0,C 180,E1 -14639.965,E2 -14639.965} C_VEL
LIN {X 0,Y 333.248,Z 346.621,A -85,B 0,C 180,E1 -14641.671,E2 -14641.671} C_VEL
LIN {X 0,Y 333.891,Z 341.079,A -85,B 0,C 180,E1 -14643.43,E2 -14643.43} C_VEL
LIN {X 0,Y 334.708,Z 334.265,A -85,B 0,C 180,E1 -14645.169,E2 -14645.169} C_VEL
LIN {X 0,Y 335.784,Z 324.94,A -85,B 0,C 180,E1 -14647.061,E2 -14647.061} C_VEL
LIN {X 0,Y 336.833,Z 315.61,A -85,B 0,C 180,E1 -14648.584,E2 -14648.584} C_VEL
LIN {X 0,Y 337.916,Z 305.172,A -85,B 0,C 180,E1 -14649.952,E2 -14649.952} C_VEL
LIN {X 0,Y 338.916,Z 294.271,A -85,B 0,C 180,E1 -14651.095,E2 -14651.095} C_VEL
LIN {X 0,Y 339.834,Z 281.635,A -85,B 0,C 180,E1 -14652.13,E2 -14652.13} C_VEL
LIN {X 0,Y 340.561,Z 268.697,A -85,B 0,C 180,E1 -14652.898,E2 -14652.898} C_VEL
LIN {X 0,Y 341.093,Z 255.571,A -85,B 0,C 180,E1 -14653.427,E2 -14653.427} C_VEL
LIN {X 0,Y 342.843,Z 173.009,A -85,B 0,C 180,E1 -14655.289,E2 -14655.289} C_VEL
LIN {X 0,Y 334.518,Z 149.465,A -85,B 0,C 180,E1 -14656.374,E2 -14656.374} C_VEL
LIN {X 0,Y 334.035,Z 147.872,A -85,B 0,C 180,E1 -14656.467,E2 -14656.467} C_VEL
LIN {X 0,Y 333.837,Z 146.903,A -85,B 0,C 180,E1 -14656.765,E2 -14656.765} C_VEL
LIN {X 0,Y 333.85,Z 146.897,A -85,B 0,C 180,E1 -14660.305,E2 -14660.305} C_VEL
LIN {X 0,Y 334.005,Z 146.877,A -85,B 0,C 180,E1 -14662.747,E2 -14662.747} C_VEL
LIN {X 0,Y 333.807,Z 146.904,A -85,B 0,C 180,E1 -14665.169,E2 -14665.169} C_VEL
LIN {X 0,Y 334.104,Z 146.868,A -85,B 0,C 180,E1 -14667.589,E2 -14667.589} C_VEL
LIN {X 0,Y 334.246,Z 146.847,A -85,B 0,C 180,E1 -14670,E2 -14670} C_VEL
LIN {X 0,Y 334.105,Z 146.864,A -85,B 0,C 180,E1 -14672.411,E2 -14672.411} C_VEL
LIN {X 0,Y 333.997,Z 146.878,A -85,B 0,C 180,E1 -14676.039,E2 -14676.039} C_VEL
LIN {X 0,Y 333.82,Z 146.901,A -85,B 0,C 180,E1 -14679.696,E2 -14679.696} C_VEL
LIN {X 0,Y 333.796,Z 146.905,A -85,B 0,C 180,E1 -14683.391,E2 -14683.391} C_VEL
LIN {X 0,Y 333.719,Z 146.916,A -85,B 0,C 180,E1 -14687.148,E2 -14687.148} C_VEL
LIN {X 0,Y 333.684,Z 146.917,A -85,B 0,C 180,E1 -14689.693,E2 -14689.693} C_VEL
LIN {X 0,Y 333.669,Z 146.919,A -85,B 0,C 180,E1 -14693.59,E2 -14693.59} C_VEL
LIN {X 0,Y 333.735,Z 146.912,A -85,B 0,C 180,E1 -14696.246,E2 -14696.246} C_VEL
LIN {X 0,Y 333.702,Z 146.916,A -85,B 0,C 180,E1 -14699.084,E2 -14699.084} C_VEL
LIN {X 0,Y 332.995,Z 147.006,A -85,B 0,C 180,E1 -14700.091,E2 -14700.091} C_VEL
LIN {X 0,Y 330.119,Z 147.361,A -85,B 0,C 180,E1 -14701.731,E2 -14701.731} C_VEL
LIN {X 0,Y 327.707,Z 147.663,A -85,B 0,C 180,E1 -14703.059,E2 -14703.059} C_VEL
LIN {X 0,Y 326.677,Z 147.792,A -85,B 0,C 180,E1 -14704.086,E2 -14704.086} C_VEL
LIN {X 0,Y 326.595,Z 147.799,A -85,B 0,C 180,E1 -14704.435,E2 -14704.435} C_VEL
LIN {X 0,Y 326.626,Z 147.796,A -85,B 0,C 180,E1 -14707.238,E2 -14707.238} C_VEL
LIN {X 0,Y 326.576,Z 147.802,A -85,B 0,C 180,E1 -14711.131,E2 -14711.131} C_VEL
LIN {X 0,Y 326.526,Z 147.81,A -85,B 0,C 180,E1 -14714.743,E2 -14714.743} C_VEL
LIN {X 0,Y 326.575,Z 147.808,A -85,B 0,C 180,E1 -14718.154,E2 -14718.154} C_VEL
LIN {X 0,Y 326.622,Z 147.796,A -85,B 0,C 180,E1 -14721.392,E2 -14721.392} C_VEL
LIN {X 0,Y 326.618,Z 147.797,A -85,B 0,C 180,E1 -14724.851,E2 -14724.851} C_VEL
LIN {X 0,Y 326.608,Z 147.8,A -85,B 0,C 180,E1 -14727.456,E2 -14727.456} C_VEL
LIN {X 0,Y 326.659,Z 147.792,A -85,B 0,C 180,E1 -14730.341,E2 -14730.341} C_VEL
LIN {X 0,Y 326.688,Z 147.788,A -85,B 0,C 180,E1 -14734.516,E2 -14734.516} C_VEL
LIN {X 0,Y 326.619,Z 147.797,A -85,B 0,C 180,E1 -14738.544,E2 -14738.544} C_VEL
LIN {X 0,Y 326.743,Z 147.783,A -85,B 0,C 180,E1 -14741.178,E2 -14741.178} C_VEL
LIN {X 0,Y 326.762,Z 147.784,A -85,B 0,C 180,E1 -14745.433,E2 -14745.433} C_VEL
LIN {X 0,Y 326.768,Z 147.779,A -85,B 0,C 180,E1 -14748.839,E2 -14748.839} C_VEL
LIN {X 0,Y 326.978,Z 147.752,A -85,B 0,C 180,E1 -14752.591,E2 -14752.591} C_VEL
LIN {X 0,Y 326.777,Z 147.78,A -85,B 0,C 180,E1 -14755.065,E2 -14755.065} C_VEL
LIN {X 0,Y 327.046,Z 147.746,A -85,B 0,C 180,E1 -14757.537,E2 -14757.537} C_VEL
LIN {X 0,Y 327.198,Z 147.725,A -85,B 0,C 180,E1 -14760,E2 -14760} C_VEL
LIN {X 0,Y 327.046,Z 147.744,A -85,B 0,C 180,E1 -14762.464,E2 -14762.464} C_VEL
LIN {X 0,Y 326.988,Z 147.751,A -85,B 0,C 180,E1 -14766.17,E2 -14766.17} C_VEL
LIN {X 0,Y 326.914,Z 147.763,A -85,B 0,C 180,E1 -14768.655,E2 -14768.655} C_VEL
LIN {X 0,Y 326.734,Z 147.784,A -85,B 0,C 180,E1 -14772.422,E2 -14772.422} C_VEL
LIN {X 0,Y 326.754,Z 147.784,A -85,B 0,C 180,E1 -14774.958,E2 -14774.958} C_VEL
LIN {X 0,Y 326.732,Z 147.786,A -85,B 0,C 180,E1 -14778.838,E2 -14778.838} C_VEL
LIN {X 0,Y 326.602,Z 147.802,A -85,B 0,C 180,E1 -14782.789,E2 -14782.789} C_VEL
LIN {X 0,Y 326.69,Z 147.788,A -85,B 0,C 180,E1 -14785.484,E2 -14785.484} C_VEL
LIN {X 0,Y 326.66,Z 147.792,A -85,B 0,C 180,E1 -14789.659,E2 -14789.659} C_VEL
LIN {X 0,Y 326.607,Z 147.802,A -85,B 0,C 180,E1 -14794.02,E2 -14794.02} C_VEL
LIN {X 0,Y 326.63,Z 147.796,A -85,B 0,C 180,E1 -14797.239,E2 -14797.239} C_VEL
LIN {X 0,Y 326.604,Z 147.803,A -85,B 0,C 180,E1 -14800.207,E2 -14800.207} C_VEL
LIN {X 0,Y 326.579,Z 147.803,A -85,B 0,C 180,E1 -14803.523,E2 -14803.523} C_VEL
LIN {X 0,Y 326.597,Z 147.8,A -85,B 0,C 180,E1 -14807.025,E2 -14807.025} C_VEL
LIN {X 0,Y 326.636,Z 147.795,A -85,B 0,C 180,E1 -14810.768,E2 -14810.768} C_VEL
LIN {X 0,Y 326.614,Z 147.798,A -85,B 0,C 180,E1 -14814.481,E2 -14814.481} C_VEL
LIN {X 0,Y 326.66,Z 147.994,A -85,B 0,C 180,E1 -14817.644,E2 -14817.644} C_VEL
LIN {X 0,Y 329.798,Z 162.212,A -85,B 0,C 180,E1 -14821.452,E2 -14821.452} C_VEL
LIN {X 0,Y 330.99,Z 168.619,A -85,B 0,C 180,E1 -14823.101,E2 -14823.101} C_VEL
LIN {X 0,Y 330.201,Z 177.268,A -85,B 0,C 180,E1 -14825.143,E2 -14825.143} C_VEL
LIN {X 0,Y 329.659,Z 182.161,A -85,B 0,C 180,E1 -14826.287,E2 -14826.287} C_VEL
LIN {X 0,Y 333.884,Z 212.411,A -85,B 0,C 180,E1 -14827.291,E2 -14827.291} C_VEL
LIN {X 0,Y 335.379,Z 225.321,A -85,B 0,C 180,E1 -14827.691,E2 -14827.691} C_VEL
LIN {X 0,Y 333.88,Z 291.842,A -85,B 0,C 180,E1 -14829.234,E2 -14829.234} C_VEL
LIN {X 0,Y 333.109,Z 305.329,A -85,B 0,C 180,E1 -14829.789,E2 -14829.789} C_VEL
LIN {X 0,Y 332.119,Z 317.638,A -85,B 0,C 180,E1 -14830.532,E2 -14830.532} C_VEL
LIN {X 0,Y 330.844,Z 330.298,A -85,B 0,C 180,E1 -14831.58,E2 -14831.58} C_VEL
LIN {X 0,Y 329.613,Z 341.612,A -85,B 0,C 180,E1 -14832.792,E2 -14832.792} C_VEL
LIN {X 0,Y 328.517,Z 351.369,A -85,B 0,C 180,E1 -14834.101,E2 -14834.101} C_VEL
LIN {X 0,Y 327.471,Z 361.027,A -85,B 0,C 180,E1 -14835.711,E2 -14835.711} C_VEL
LIN {X 0,Y 326.415,Z 369.995,A -85,B 0,C 180,E1 -14837.566,E2 -14837.566} C_VEL
LIN {X 0,Y 325.671,Z 377.172,A -85,B 0,C 180,E1 -14839.43,E2 -14839.43} C_VEL
LIN {X 0,Y 325.28,Z 382.89,A -85,B 0,C 180,E1 -14841.301,E2 -14841.301} C_VEL
LIN {X 0,Y 325.046,Z 387.367,A -85,B 0,C 180,E1 -14843.17,E2 -14843.17} C_VEL
LIN {X 0,Y 324.973,Z 390.73,A -85,B 0,C 180,E1 -14845.037,E2 -14845.037} C_VEL
LIN {X 0,Y 324.993,Z 392.39,A -85,B 0,C 180,E1 -14846.28,E2 -14846.28} C_VEL
LIN {X 0,Y 324.995,Z 393.63,A -85,B 0,C 180,E1 -14847.521,E2 -14847.521} C_VEL
LIN {X 0,Y 325.111,Z 394.451,A -85,B 0,C 180,E1 -14848.761,E2 -14848.761} C_VEL
LIN {X 0,Y 325.174,Z 394.82,A -85,B 0,C 180,E1 -14850,E2 -14850} C_VEL
LIN {X 0,Y 325.065,Z 394.78,A -85,B 0,C 180,E1 -14851.239,E2 -14851.239} C_VEL
LIN {X 0,Y 324.956,Z 394.345,A -85,B 0,C 180,E1 -14852.479,E2 -14852.479} C_VEL
LIN {X 0,Y 324.971,Z 393.504,A -85,B 0,C 180,E1 -14853.72,E2 -14853.72} C_VEL
LIN {X 0,Y 324.918,Z 391.22,A -85,B 0,C 180,E1 -14855.737,E2 -14855.737} C_VEL
LIN {X 0,Y 325.179,Z 387.125,A -85,B 0,C 180,E1 -14858.076,E2 -14858.076} C_VEL
LIN {X 0,Y 325.573,Z 382.662,A -85,B 0,C 180,E1 -14859.944,E2 -14859.944} C_VEL
LIN {X 0,Y 326.252,Z 377.007,A -85,B 0,C 180,E1 -14861.809,E2 -14861.809} C_VEL
LIN {X 0,Y 327.349,Z 369.983,A -85,B 0,C 180,E1 -14863.66,E2 -14863.66} C_VEL
LIN {X 0,Y 328.505,Z 362.148,A -85,B 0,C 180,E1 -14865.334,E2 -14865.334} C_VEL
LIN {X 0,Y 329.89,Z 352.302,A -85,B 0,C 180,E1 -14867.033,E2 -14867.033} C_VEL
LIN {X 0,Y 331.525,Z 341.376,A -85,B 0,C 180,E1 -14868.541,E2 -14868.541} C_VEL
LIN {X 0,Y 333.091,Z 330.42,A -85,B 0,C 180,E1 -14869.73,E2 -14869.73} C_VEL
LIN {X 0,Y 334.566,Z 318.23,A -85,B 0,C 180,E1 -14870.761,E2 -14870.761} C_VEL
LIN {X 0,Y 335.909,Z 305.55,A -85,B 0,C 180,E1 -14871.558,E2 -14871.558} C_VEL
LIN {X 0,Y 336.861,Z 292.353,A -85,B 0,C 180,E1 -14872.126,E2 -14872.126} C_VEL
LIN {X 0,Y 337.528,Z 272.71,A -85,B 0,C 180,E1 -14872.629,E2 -14872.629} C_VEL
LIN {X 0,Y 338.676,Z 223.693,A -85,B 0,C 180,E1 -14873.775,E2 -14873.775} C_VEL
LIN {X 0,Y 335.675,Z 202.114,A -85,B 0,C 180,E1 -14874.596,E2 -14874.596} C_VEL
LIN {X 0,Y 331.445,Z 179.692,A -85,B 0,C 180,E1 -14875.613,E2 -14875.613} C_VEL
LIN {X 0,Y 332.245,Z 172.532,A -85,B 0,C 180,E1 -14877.323,E2 -14877.323} C_VEL
LIN {X 0,Y 330.308,Z 162.73,A -85,B 0,C 180,E1 -14880,E2 -14880} C_VEL
LIN {X 0,Y 327.927,Z 152.742,A -85,B 0,C 180,E1 -14882.908,E2 -14882.908} C_VEL
LIN {X 0,Y 326.638,Z 147.803,A -85,B 0,C 180,E1 -14884.481,E2 -14884.481} C_VEL
LIN {X 0,Y 326.644,Z 147.802,A -85,B 0,C 180,E1 -14888.605,E2 -14888.605} C_VEL
LIN {X 0,Y 326.596,Z 147.808,A -85,B 0,C 180,E1 -14891.842,E2 -14891.842} C_VEL
LIN {X 0,Y 326.546,Z 147.812,A -85,B 0,C 180,E1 -14895.254,E2 -14895.254} C_VEL
LIN {X 0,Y 326.592,Z 147.803,A -85,B 0,C 180,E1 -14898.865,E2 -14898.865} C_VEL
LIN {X 0,Y 326.643,Z 147.793,A -85,B 0,C 180,E1 -14901.394,E2 -14901.394} C_VEL
LIN {X 0,Y 326.619,Z 147.798,A -85,B 0,C 180,E1 -14904.851,E2 -14904.851} C_VEL
LIN {X 0,Y 326.607,Z 147.796,A -85,B 0,C 180,E1 -14907.455,E2 -14907.455} C_VEL
LIN {X 0,Y 326.66,Z 147.788,A -85,B 0,C 180,E1 -14910.341,E2 -14910.341} C_VEL
LIN {X 0,Y 326.689,Z 147.785,A -85,B 0,C 180,E1 -14914.516,E2 -14914.516} C_VEL
LIN {X 0,Y 326.619,Z 147.795,A -85,B 0,C 180,E1 -14918.543,E2 -14918.543} C_VEL
LIN {X 0,Y 326.743,Z 147.775,A -85,B 0,C 180,E1 -14921.177,E2 -14921.177} C_VEL
LIN {X 0,Y 326.762,Z 147.775,A -85,B 0,C 180,E1 -14925.433,E2 -14925.433} C_VEL
LIN {X 0,Y 326.768,Z 147.774,A -85,B 0,C 180,E1 -14928.839,E2 -14928.839} C_VEL
LIN {X 0,Y 326.978,Z 147.748,A -85,B 0,C 180,E1 -14932.59,E2 -14932.59} C_VEL
LIN {X 0,Y 326.776,Z 147.779,A -85,B 0,C 180,E1 -14935.065,E2 -14935.065} C_VEL
LIN {X 0,Y 327.046,Z 147.748,A -85,B 0,C 180,E1 -14937.536,E2 -14937.536} C_VEL
LIN {X 0,Y 327.197,Z 147.722,A -85,B 0,C 180,E1 -14940,E2 -14940} C_VEL
LIN {X 0,Y 327.046,Z 147.745,A -85,B 0,C 180,E1 -14942.463,E2 -14942.463} C_VEL
LIN {X 0,Y 326.959,Z 147.752,A -85,B 0,C 180,E1 -14946.587,E2 -14946.587} C_VEL
LIN {X 0,Y 326.804,Z 147.777,A -85,B 0,C 180,E1 -14949.906,E2 -14949.906} C_VEL
LIN {X 0,Y 326.757,Z 147.781,A -85,B 0,C 180,E1 -14953.685,E2 -14953.685} C_VEL
LIN {X 0,Y 326.697,Z 147.79,A -85,B 0,C 180,E1 -14957.528,E2 -14957.528} C_VEL
LIN {X 0,Y 326.663,Z 147.795,A -85,B 0,C 180,E1 -14960.135,E2 -14960.135} C_VEL
LIN {X 0,Y 326.65,Z 147.803,A -85,B 0,C 180,E1 -14964.129,E2 -14964.129} C_VEL
LIN {X 0,Y 326.687,Z 147.849,A -85,B 0,C 180,E1 -14966.168,E2 -14966.168} C_VEL
LIN {X 0,Y 327.345,Z 150.497,A -85,B 0,C 180,E1 -14967.058,E2 -14967.058} C_VEL
LIN {X 0,Y 335.151,Z 166.982,A -85,B 0,C 180,E1 -14968.284,E2 -14968.284} C_VEL
LIN {X 0,Y 339.885,Z 178.514,A -85,B 0,C 180,E1 -14969.03,E2 -14969.03} C_VEL
LIN {X 0,Y 337.649,Z 257.905,A -85,B 0,C 180,E1 -14970.902,E2 -14970.902} C_VEL
LIN {X 0,Y 336.931,Z 271.443,A -85,B 0,C 180,E1 -14971.475,E2 -14971.475} C_VEL
LIN {X 0,Y 336.093,Z 283.479,A -85,B 0,C 180,E1 -14972.224,E2 -14972.224} C_VEL
LIN {X 0,Y 335.001,Z 294.903,A -85,B 0,C 180,E1 -14973.173,E2 -14973.173} C_VEL
LIN {X 0,Y 333.632,Z 306.428,A -85,B 0,C 180,E1 -14974.401,E2 -14974.401} C_VEL
LIN {X 0,Y 332.264,Z 316.44,A -85,B 0,C 180,E1 -14975.738,E2 -14975.738} C_VEL
LIN {X 0,Y 330.892,Z 325.336,A -85,B 0,C 180,E1 -14977.205,E2 -14977.205} C_VEL
LIN {X 0,Y 329.504,Z 333.557,A -85,B 0,C 180,E1 -14978.876,E2 -14978.876} C_VEL
LIN {X 0,Y 328.282,Z 340.565,A -85,B 0,C 180,E1 -14980.636,E2 -14980.636} C_VEL
LIN {X 0,Y 327.358,Z 346.105,A -85,B 0,C 180,E1 -14982.363,E2 -14982.363} C_VEL
LIN {X 0,Y 326.616,Z 350.549,A -85,B 0,C 180,E1 -14984.095,E2 -14984.095} C_VEL
LIN {X 0,Y 325.858,Z 354.906,A -85,B 0,C 180,E1 -14986.357,E2 -14986.357} C_VEL
LIN {X 0,Y 325.442,Z 357.071,A -85,B 0,C 180,E1 -14987.976,E2 -14987.976} C_VEL
LIN {X 0,Y 325.141,Z 358.535,A -85,B 0,C 180,E1 -14989.575,E2 -14989.575} C_VEL
LIN {X 0,Y 324.986,Z 359.298,A -85,B 0,C 180,E1 -14991.161,E2 -14991.161} C_VEL
LIN {X 0,Y 324.887,Z 359.334,A -85,B 0,C 180,E1 -14993.167,E2 -14993.167} C_VEL
LIN {X 0,Y 324.956,Z 358.254,A -85,B 0,C 180,E1 -14995.27,E2 -14995.27} C_VEL
LIN {X 0,Y 325.26,Z 355.906,A -85,B 0,C 180,E1 -14997.424,E2 -14997.424} C_VEL
LIN {X 0,Y 325.677,Z 352.042,A -85,B 0,C 180,E1 -14999.676,E2 -14999.676} C_VEL
LIN {X 0,Y 326.187,Z 347.226,A -85,B 0,C 180,E1 -15001.705,E2 -15001.705} C_VEL
LIN {X 0,Y 326.99,Z 340.567,A -85,B 0,C 180,E1 -15003.838,E2 -15003.838} C_VEL
LIN {X 0,Y 327.828,Z 333.464,A -85,B 0,C 180,E1 -15005.627,E2 -15005.627} C_VEL
LIN {X 0,Y 328.894,Z 324.841,A -85,B 0,C 180,E1 -15007.379,E2 -15007.379} C_VEL
LIN {X 0,Y 330.016,Z 315.214,A -85,B 0,C 180,E1 -15008.958,E2 -15008.958} C_VEL
LIN {X 0,Y 331.1,Z 304.955,A -85,B 0,C 180,E1 -15010.308,E2 -15010.308} C_VEL
LIN {X 0,Y 332.169,Z 293.676,A -85,B 0,C 180,E1 -15011.496,E2 -15011.496} C_VEL
LIN {X 0,Y 333,Z 282.224,A -85,B 0,C 180,E1 -15012.445,E2 -15012.445} C_VEL
LIN {X 0,Y 333.765,Z 269.726,A -85,B 0,C 180,E1 -15013.21,E2 -15013.21} C_VEL
LIN {X 0,Y 334.311,Z 256.384,A -85,B 0,C 180,E1 -15013.768,E2 -15013.768} C_VEL
LIN {X 0,Y 336.158,Z 174.39,A -85,B 0,C 180,E1 -15015.664,E2 -15015.664} C_VEL
LIN {X 0,Y 327.611,Z 150.44,A -85,B 0,C 180,E1 -15016.805,E2 -15016.805} C_VEL
LIN {X 0,Y 326.84,Z 148.185,A -85,B 0,C 180,E1 -15016.951,E2 -15016.951} C_VEL
LIN {X 0,Y 326.803,Z 147.78,A -85,B 0,C 180,E1 -15017.108,E2 -15017.108} C_VEL
LIN {X 0,Y 326.922,Z 147.765,A -85,B 0,C 180,E1 -15021.448,E2 -15021.448} C_VEL
LIN {X 0,Y 326.988,Z 147.754,A -85,B 0,C 180,E1 -15023.831,E2 -15023.831} C_VEL
LIN {X 0,Y 327.045,Z 147.748,A -85,B 0,C 180,E1 -15027.537,E2 -15027.537} C_VEL
LIN {X 0,Y 327.197,Z 147.726,A -85,B 0,C 180,E1 -15030,E2 -15030} C_VEL
LIN {X 0,Y 327.045,Z 147.744,A -85,B 0,C 180,E1 -15032.463,E2 -15032.463} C_VEL
LIN {X 0,Y 326.951,Z 147.756,A -85,B 0,C 180,E1 -15036.17,E2 -15036.17} C_VEL
LIN {X 0,Y 326.783,Z 147.777,A -85,B 0,C 180,E1 -15039.907,E2 -15039.907} C_VEL
LIN {X 0,Y 326.759,Z 147.78,A -85,B 0,C 180,E1 -15043.685,E2 -15043.685} C_VEL
LIN {X 0,Y 326.663,Z 147.792,A -85,B 0,C 180,E1 -15047.53,E2 -15047.53} C_VEL
LIN {X 0,Y 326.63,Z 147.796,A -85,B 0,C 180,E1 -15050.137,E2 -15050.137} C_VEL
LIN {X 0,Y 326.648,Z 147.794,A -85,B 0,C 180,E1 -15054.129,E2 -15054.129} C_VEL
LIN {X 0,Y 326.684,Z 147.793,A -85,B 0,C 180,E1 -15056.858,E2 -15056.858} C_VEL
LIN {X 0,Y 326.638,Z 147.8,A -85,B 0,C 180,E1 -15060.611,E2 -15060.611} C_VEL
LIN {X 0,Y 326.595,Z 147.799,A -85,B 0,C 180,E1 -15064.435,E2 -15064.435} C_VEL
LIN {X 0,Y 325.943,Z 147.882,A -85,B 0,C 180,E1 -15065.464,E2 -15065.464} C_VEL
LIN {X 0,Y 323.125,Z 148.235,A -85,B 0,C 180,E1 -15067.141,E2 -15067.141} C_VEL
LIN {X 0,Y 320.711,Z 148.537,A -85,B 0,C 180,E1 -15068.5,E2 -15068.5} C_VEL
LIN {X 0,Y 319.641,Z 148.666,A -85,B 0,C 180,E1 -15069.55,E2 -15069.55} C_VEL
LIN {X 0,Y 319.537,Z 148.677,A -85,B 0,C 180,E1 -15069.907,E2 -15069.907} C_VEL
LIN {X 0,Y 319.52,Z 148.681,A -85,B 0,C 180,E1 -15073.461,E2 -15073.461} C_VEL
LIN {X 0,Y 319.552,Z 148.677,A -85,B 0,C 180,E1 -15077.017,E2 -15077.017} C_VEL
LIN {X 0,Y 319.546,Z 148.68,A -85,B 0,C 180,E1 -15080.371,E2 -15080.371} C_VEL
LIN {X 0,Y 319.557,Z 148.678,A -85,B 0,C 180,E1 -15083.573,E2 -15083.573} C_VEL
LIN {X 0,Y 319.576,Z 148.674,A -85,B 0,C 180,E1 -15086.686,E2 -15086.686} C_VEL
LIN {X 0,Y 319.59,Z 148.675,A -85,B 0,C 180,E1 -15089.617,E2 -15089.617} C_VEL
LIN {X 0,Y 319.607,Z 148.67,A -85,B 0,C 180,E1 -15092.498,E2 -15092.498} C_VEL
LIN {X 0,Y 319.601,Z 148.673,A -85,B 0,C 180,E1 -15095.304,E2 -15095.304} C_VEL
LIN {X 0,Y 319.602,Z 148.674,A -85,B 0,C 180,E1 -15099.401,E2 -15099.401} C_VEL
LIN {X 0,Y 319.657,Z 148.664,A -85,B 0,C 180,E1 -15102.073,E2 -15102.073} C_VEL
LIN {X 0,Y 319.731,Z 148.656,A -85,B 0,C 180,E1 -15106.008,E2 -15106.008} C_VEL
LIN {X 0,Y 319.756,Z 148.653,A -85,B 0,C 180,E1 -15109.873,E2 -15109.873} C_VEL
LIN {X 0,Y 319.932,Z 148.629,A -85,B 0,C 180,E1 -15112.426,E2 -15112.426} C_VEL
LIN {X 0,Y 319.746,Z 148.654,A -85,B 0,C 180,E1 -15114.956,E2 -15114.956} C_VEL
LIN {X 0,Y 319.99,Z 148.625,A -85,B 0,C 180,E1 -15117.483,E2 -15117.483} C_VEL
LIN {X 0,Y 320.149,Z 148.602,A -85,B 0,C 180,E1 -15120,E2 -15120} C_VEL
LIN {X 0,Y 319.99,Z 148.623,A -85,B 0,C 180,E1 -15122.518,E2 -15122.518} C_VEL
LIN {X 0,Y 319.944,Z 148.629,A -85,B 0,C 180,E1 -15126.306,E2 -15126.306} C_VEL
LIN {X 0,Y 319.842,Z 148.646,A -85,B 0,C 180,E1 -15128.848,E2 -15128.848} C_VEL
LIN {X 0,Y 319.681,Z 148.665,A -85,B 0,C 180,E1 -15132.7,E2 -15132.7} C_VEL
LIN {X 0,Y 319.699,Z 148.66,A -85,B 0,C 180,E1 -15135.296,E2 -15135.296} C_VEL
LIN {X 0,Y 319.673,Z 148.662,A -85,B 0,C 180,E1 -15139.255,E2 -15139.255} C_VEL
LIN {X 0,Y 319.56,Z 148.677,A -85,B 0,C 180,E1 -15143.321,E2 -15143.321} C_VEL
LIN {X 0,Y 319.634,Z 148.669,A -85,B 0,C 180,E1 -15146.088,E2 -15146.088} C_VEL
LIN {X 0,Y 319.589,Z 148.674,A -85,B 0,C 180,E1 -15148.934,E2 -15148.934} C_VEL
LIN {X 0,Y 319.532,Z 148.681,A -85,B 0,C 180,E1 -15151.862,E2 -15151.862} C_VEL
LIN {X 0,Y 319.58,Z 148.675,A -85,B 0,C 180,E1 -15155.543,E2 -15155.543} C_VEL
LIN {X 0,Y 319.598,Z 148.676,A -85,B 0,C 180,E1 -15158.005,E2 -15158.005} C_VEL
LIN {X 0,Y 319.567,Z 148.677,A -85,B 0,C 180,E1 -15161.606,E2 -15161.606} C_VEL
LIN {X 0,Y 319.503,Z 148.684,A -85,B 0,C 180,E1 -15165.26,E2 -15165.26} C_VEL
LIN {X 0,Y 319.544,Z 148.679,A -85,B 0,C 180,E1 -15168.714,E2 -15168.714} C_VEL
LIN {X 0,Y 319.583,Z 148.675,A -85,B 0,C 180,E1 -15172.343,E2 -15172.343} C_VEL
LIN {X 0,Y 319.562,Z 148.678,A -85,B 0,C 180,E1 -15175.124,E2 -15175.124} C_VEL
LIN {X 0,Y 319.607,Z 148.805,A -85,B 0,C 180,E1 -15177.262,E2 -15177.262} C_VEL
LIN {X 0,Y 322.519,Z 162.09,A -85,B 0,C 180,E1 -15180.913,E2 -15180.913} C_VEL
LIN {X 0,Y 323.981,Z 169.626,A -85,B 0,C 180,E1 -15182.9,E2 -15182.9} C_VEL
LIN {X 0,Y 323.585,Z 175.192,A -85,B 0,C 180,E1 -15184.254,E2 -15184.254} C_VEL
LIN {X 0,Y 322.831,Z 181.735,A -85,B 0,C 180,E1 -15185.819,E2 -15185.819} C_VEL
LIN {X 0,Y 327.031,Z 211.92,A -85,B 0,C 180,E1 -15186.864,E2 -15186.864} C_VEL
LIN {X 0,Y 328.655,Z 226.098,A -85,B 0,C 180,E1 -15187.315,E2 -15187.315} C_VEL
LIN {X 0,Y 327.115,Z 291.542,A -85,B 0,C 180,E1 -15188.867,E2 -15188.867} C_VEL
LIN {X 0,Y 326.316,Z 304.993,A -85,B 0,C 180,E1 -15189.431,E2 -15189.431} C_VEL
LIN {X 0,Y 325.302,Z 317.287,A -85,B 0,C 180,E1 -15190.189,E2 -15190.189} C_VEL
LIN {X 0,Y 324.074,Z 329.146,A -85,B 0,C 180,E1 -15191.181,E2 -15191.181} C_VEL
LIN {X 0,Y 322.759,Z 340.594,A -85,B 0,C 180,E1 -15192.415,E2 -15192.415} C_VEL
LIN {X 0,Y 321.648,Z 350.229,A -85,B 0,C 180,E1 -15193.714,E2 -15193.714} C_VEL
LIN {X 0,Y 320.729,Z 358.541,A -85,B 0,C 180,E1 -15195.08,E2 -15195.08} C_VEL
LIN {X 0,Y 319.808,Z 366.519,A -85,B 0,C 180,E1 -15196.659,E2 -15196.659} C_VEL
LIN {X 0,Y 318.841,Z 374.277,A -85,B 0,C 180,E1 -15198.558,E2 -15198.558} C_VEL
LIN {X 0,Y 318.315,Z 380.512,A -85,B 0,C 180,E1 -15200.468,E2 -15200.468} C_VEL
LIN {X 0,Y 318.023,Z 385.442,A -85,B 0,C 180,E1 -15202.38,E2 -15202.38} C_VEL
LIN {X 0,Y 317.918,Z 388.97,A -85,B 0,C 180,E1 -15204.15,E2 -15204.15} C_VEL
LIN {X 0,Y 317.918,Z 391.918,A -85,B 0,C 180,E1 -15206.197,E2 -15206.197} C_VEL
LIN {X 0,Y 317.907,Z 393.176,A -85,B 0,C 180,E1 -15207.466,E2 -15207.466} C_VEL
LIN {X 0,Y 318.015,Z 394.026,A -85,B 0,C 180,E1 -15208.734,E2 -15208.734} C_VEL
LIN {X 0,Y 318.083,Z 394.42,A -85,B 0,C 180,E1 -15210,E2 -15210} C_VEL
LIN {X 0,Y 317.969,Z 394.397,A -85,B 0,C 180,E1 -15211.266,E2 -15211.266} C_VEL
LIN {X 0,Y 317.894,Z 393.163,A -85,B 0,C 180,E1 -15213.803,E2 -15213.803} C_VEL
LIN {X 0,Y 317.821,Z 391.157,A -85,B 0,C 180,E1 -15215.678,E2 -15215.678} C_VEL
LIN {X 0,Y 318.009,Z 388.099,A -85,B 0,C 180,E1 -15217.62,E2 -15217.62} C_VEL
LIN {X 0,Y 318.36,Z 384.04,A -85,B 0,C 180,E1 -15219.53,E2 -15219.53} C_VEL
LIN {X 0,Y 319.124,Z 377.848,A -85,B 0,C 180,E1 -15221.754,E2 -15221.754} C_VEL
LIN {X 0,Y 320.218,Z 371.108,A -85,B 0,C 180,E1 -15223.647,E2 -15223.647} C_VEL
LIN {X 0,Y 321.55,Z 362.682,A -85,B 0,C 180,E1 -15225.55,E2 -15225.55} C_VEL
LIN {X 0,Y 322.79,Z 354.294,A -85,B 0,C 180,E1 -15227.093,E2 -15227.093} C_VEL
LIN {X 0,Y 324.416,Z 343.888,A -85,B 0,C 180,E1 -15228.635,E2 -15228.635} C_VEL
LIN {X 0,Y 326.238,Z 332.21,A -85,B 0,C 180,E1 -15229.998,E2 -15229.998} C_VEL
LIN {X 0,Y 327.769,Z 320.717,A -85,B 0,C 180,E1 -15231.048,E2 -15231.048} C_VEL
LIN {X 0,Y 329.198,Z 307.646,A -85,B 0,C 180,E1 -15231.938,E2 -15231.938} C_VEL
LIN {X 0,Y 330.283,Z 294.757,A -85,B 0,C 180,E1 -15232.557,E2 -15232.557} C_VEL
LIN {X 0,Y 330.901,Z 281.656,A -85,B 0,C 180,E1 -15232.952,E2 -15232.952} C_VEL
LIN {X 0,Y 332.419,Z 225.116,A -85,B 0,C 180,E1 -15234.289,E2 -15234.289} C_VEL
LIN {X 0,Y 329.516,Z 203.859,A -85,B 0,C 180,E1 -15235.13,E2 -15235.13} C_VEL
LIN {X 0,Y 325.263,Z 181.543,A -85,B 0,C 180,E1 -15236.159,E2 -15236.159} C_VEL
LIN {X 0,Y 324.813,Z 179.265,A -85,B 0,C 180,E1 -15236.282,E2 -15236.282} C_VEL
LIN {X 0,Y 325.337,Z 173.662,A -85,B 0,C 180,E1 -15237.663,E2 -15237.663} C_VEL
LIN {X 0,Y 323.443,Z 164.152,A -85,B 0,C 180,E1 -15240.344,E2 -15240.344} C_VEL
LIN {X 0,Y 321.163,Z 154.735,A -85,B 0,C 180,E1 -15243.166,E2 -15243.166} C_VEL
LIN {X 0,Y 319.602,Z 148.677,A -85,B 0,C 180,E1 -15245.121,E2 -15245.121} C_VEL
LIN {X 0,Y 319.599,Z 148.683,A -85,B 0,C 180,E1 -15248.004,E2 -15248.004} C_VEL
LIN {X 0,Y 319.567,Z 148.682,A -85,B 0,C 180,E1 -15251.605,E2 -15251.605} C_VEL
LIN {X 0,Y 319.505,Z 148.689,A -85,B 0,C 180,E1 -15255.26,E2 -15255.26} C_VEL
LIN {X 0,Y 319.544,Z 148.68,A -85,B 0,C 180,E1 -15258.714,E2 -15258.714} C_VEL
LIN {X 0,Y 319.597,Z 148.676,A -85,B 0,C 180,E1 -15262.339,E2 -15262.339} C_VEL
LIN {X 0,Y 319.56,Z 148.678,A -85,B 0,C 180,E1 -15265.123,E2 -15265.123} C_VEL
LIN {X 0,Y 319.57,Z 148.678,A -85,B 0,C 180,E1 -15269.057,E2 -15269.057} C_VEL
LIN {X 0,Y 319.608,Z 148.671,A -85,B 0,C 180,E1 -15272.498,E2 -15272.498} C_VEL
LIN {X 0,Y 319.602,Z 148.671,A -85,B 0,C 180,E1 -15275.303,E2 -15275.303} C_VEL
LIN {X 0,Y 319.603,Z 148.673,A -85,B 0,C 180,E1 -15279.4,E2 -15279.4} C_VEL
LIN {X 0,Y 319.657,Z 148.663,A -85,B 0,C 180,E1 -15282.073,E2 -15282.073} C_VEL
LIN {X 0,Y 319.731,Z 148.657,A -85,B 0,C 180,E1 -15286.007,E2 -15286.007} C_VEL
LIN {X 0,Y 319.756,Z 148.654,A -85,B 0,C 180,E1 -15289.873,E2 -15289.873} C_VEL
LIN {X 0,Y 319.932,Z 148.625,A -85,B 0,C 180,E1 -15292.426,E2 -15292.426} C_VEL
LIN {X 0,Y 319.746,Z 148.656,A -85,B 0,C 180,E1 -15294.956,E2 -15294.956} C_VEL
LIN {X 0,Y 319.989,Z 148.627,A -85,B 0,C 180,E1 -15297.482,E2 -15297.482} C_VEL
LIN {X 0,Y 320.149,Z 148.6,A -85,B 0,C 180,E1 -15300,E2 -15300} C_VEL
LIN {X 0,Y 319.989,Z 148.623,A -85,B 0,C 180,E1 -15302.517,E2 -15302.517} C_VEL
LIN {X 0,Y 319.921,Z 148.629,A -85,B 0,C 180,E1 -15306.574,E2 -15306.574} C_VEL
LIN {X 0,Y 319.751,Z 148.656,A -85,B 0,C 180,E1 -15310.127,E2 -15310.127} C_VEL
LIN {X 0,Y 319.729,Z 148.659,A -85,B 0,C 180,E1 -15314.724,E2 -15314.724} C_VEL
LIN {X 0,Y 319.687,Z 148.665,A -85,B 0,C 180,E1 -15319.038,E2 -15319.038} C_VEL
LIN {X 0,Y 319.568,Z 148.684,A -85,B 0,C 180,E1 -15323.319,E2 -15323.319} C_VEL
LIN {X 0,Y 319.663,Z 148.739,A -85,B 0,C 180,E1 -15325.516,E2 -15325.516} C_VEL
LIN {X 0,Y 320.223,Z 150.995,A -85,B 0,C 180,E1 -15326.299,E2 -15326.299} C_VEL
LIN {X 0,Y 327.234,Z 165.371,A -85,B 0,C 180,E1 -15327.457,E2 -15327.457} C_VEL
LIN {X 0,Y 333.33,Z 179.556,A -85,B 0,C 180,E1 -15328.445,E2 -15328.445} C_VEL
LIN {X 0,Y 333.714,Z 180.628,A -85,B 0,C 180,E1 -15328.51,E2 -15328.51} C_VEL
LIN {X 0,Y 331.262,Z 258.615,A -85,B 0,C 180,E1 -15330.386,E2 -15330.386} C_VEL
LIN {X 0,Y 330.5,Z 272.224,A -85,B 0,C 180,E1 -15330.979,E2 -15330.979} C_VEL
LIN {X 0,Y 329.692,Z 283.323,A -85,B 0,C 180,E1 -15331.681,E2 -15331.681} C_VEL
LIN {X 0,Y 328.526,Z 295.038,A -85,B 0,C 180,E1 -15332.66,E2 -15332.66} C_VEL
LIN {X 0,Y 327.121,Z 306.445,A -85,B 0,C 180,E1 -15333.89,E2 -15333.89} C_VEL
LIN {X 0,Y 325.66,Z 316.689,A -85,B 0,C 180,E1 -15335.276,E2 -15335.276} C_VEL
LIN {X 0,Y 324.077,Z 326.347,A -85,B 0,C 180,E1 -15336.909,E2 -15336.909} C_VEL
LIN {X 0,Y 322.616,Z 334.554,A -85,B 0,C 180,E1 -15338.633,E2 -15338.633} C_VEL
LIN {X 0,Y 321.226,Z 342.161,A -85,B 0,C 180,E1 -15340.631,E2 -15340.631} C_VEL
LIN {X 0,Y 320.282,Z 347.484,A -85,B 0,C 180,E1 -15342.403,E2 -15342.403} C_VEL
LIN {X 0,Y 319.516,Z 351.768,A -85,B 0,C 180,E1 -15344.199,E2 -15344.199} C_VEL
LIN {X 0,Y 318.89,Z 355.068,A -85,B 0,C 180,E1 -15345.998,E2 -15345.998} C_VEL
LIN {X 0,Y 318.244,Z 358.194,A -85,B 0,C 180,E1 -15348.509,E2 -15348.509} C_VEL
LIN {X 0,Y 317.928,Z 359.571,A -85,B 0,C 180,E1 -15350.687,E2 -15350.687} C_VEL
LIN {X 0,Y 317.802,Z 359.785,A -85,B 0,C 180,E1 -15352.761,E2 -15352.761} C_VEL
LIN {X 0,Y 317.849,Z 358.875,A -85,B 0,C 180,E1 -15354.908,E2 -15354.908} C_VEL
LIN {X 0,Y 318.102,Z 356.757,A -85,B 0,C 180,E1 -15357.093,E2 -15357.093} C_VEL
LIN {X 0,Y 318.54,Z 352.923,A -85,B 0,C 180,E1 -15359.506,E2 -15359.506} C_VEL
LIN {X 0,Y 319.109,Z 347.79,A -85,B 0,C 180,E1 -15361.757,E2 -15361.757} C_VEL
LIN {X 0,Y 319.958,Z 341.175,A -85,B 0,C 180,E1 -15363.941,E2 -15363.941} C_VEL
LIN {X 0,Y 320.804,Z 334.209,A -85,B 0,C 180,E1 -15365.747,E2 -15365.747} C_VEL
LIN {X 0,Y 321.9,Z 325.648,A -85,B 0,C 180,E1 -15367.538,E2 -15367.538} C_VEL
LIN {X 0,Y 323.001,Z 316.444,A -85,B 0,C 180,E1 -15369.102,E2 -15369.102} C_VEL
LIN {X 0,Y 324.148,Z 306.016,A -85,B 0,C 180,E1 -15370.528,E2 -15370.528} C_VEL
LIN {X 0,Y 325.269,Z 294.705,A -85,B 0,C 180,E1 -15371.758,E2 -15371.758} C_VEL
LIN {X 0,Y 326.179,Z 282.892,A -85,B 0,C 180,E1 -15372.767,E2 -15372.767} C_VEL
LIN {X 0,Y 326.966,Z 270.782,A -85,B 0,C 180,E1 -15373.533,E2 -15373.533} C_VEL
LIN {X 0,Y 327.523,Z 257.331,A -85,B 0,C 180,E1 -15374.119,E2 -15374.119} C_VEL
LIN {X 0,Y 328.45,Z 220.749,A -85,B 0,C 180,E1 -15375.003,E2 -15375.003} C_VEL
LIN {X 0,Y 329.495,Z 175.939,A -85,B 0,C 180,E1 -15376.044,E2 -15376.044} C_VEL
LIN {X 0,Y 321.295,Z 153.024,A -85,B 0,C 180,E1 -15377.166,E2 -15377.166} C_VEL
LIN {X 0,Y 319.729,Z 148.66,A -85,B 0,C 180,E1 -15377.423,E2 -15377.423} C_VEL
LIN {X 0,Y 319.877,Z 148.642,A -85,B 0,C 180,E1 -15381.374,E2 -15381.374} C_VEL
LIN {X 0,Y 319.943,Z 148.633,A -85,B 0,C 180,E1 -15383.694,E2 -15383.694} C_VEL
LIN {X 0,Y 319.989,Z 148.628,A -85,B 0,C 180,E1 -15387.482,E2 -15387.482} C_VEL
LIN {X 0,Y 320.149,Z 148.604,A -85,B 0,C 180,E1 -15390,E2 -15390} C_VEL
LIN {X 0,Y 319.989,Z 148.623,A -85,B 0,C 180,E1 -15392.518,E2 -15392.518} C_VEL
LIN {X 0,Y 319.907,Z 148.633,A -85,B 0,C 180,E1 -15396.306,E2 -15396.306} C_VEL
LIN {X 0,Y 319.735,Z 148.655,A -85,B 0,C 180,E1 -15400.128,E2 -15400.128} C_VEL
LIN {X 0,Y 319.732,Z 148.655,A -85,B 0,C 180,E1 -15403.992,E2 -15403.992} C_VEL
LIN {X 0,Y 319.624,Z 148.668,A -85,B 0,C 180,E1 -15407.929,E2 -15407.929} C_VEL
LIN {X 0,Y 319.567,Z 148.675,A -85,B 0,C 180,E1 -15411.954,E2 -15411.954} C_VEL
LIN {X 0,Y 319.634,Z 148.668,A -85,B 0,C 180,E1 -15416.088,E2 -15416.088} C_VEL
LIN {X 0,Y 319.589,Z 148.675,A -85,B 0,C 180,E1 -15418.934,E2 -15418.934} C_VEL
LIN {X 0,Y 319.531,Z 148.68,A -85,B 0,C 180,E1 -15421.862,E2 -15421.862} C_VEL
LIN {X 0,Y 319.578,Z 148.674,A -85,B 0,C 180,E1 -15425.543,E2 -15425.543} C_VEL
LIN {X 0,Y 319.556,Z 148.679,A -85,B 0,C 180,E1 -15428.01,E2 -15428.01} C_VEL
LIN {X 0,Y 319.537,Z 148.677,A -85,B 0,C 180,E1 -15429.907,E2 -15429.907} C_VEL
LIN {X 0,Y 318.811,Z 148.77,A -85,B 0,C 180,E1 -15430.958,E2 -15430.958} C_VEL
LIN {X 0,Y 315.907,Z 149.133,A -85,B 0,C 180,E1 -15432.668,E2 -15432.668} C_VEL
LIN {X 0,Y 313.498,Z 149.435,A -85,B 0,C 180,E1 -15434.054,E2 -15434.054} C_VEL
LIN {X 0,Y 312.497,Z 149.556,A -85,B 0,C 180,E1 -15435.128,E2 -15435.128} C_VEL
LIN {X 0,Y 312.432,Z 149.564,A -85,B 0,C 180,E1 -15435.491,E2 -15435.491} C_VEL
LIN {X 0,Y 312.488,Z 149.556,A -85,B 0,C 180,E1 -15439.291,E2 -15439.291} C_VEL
LIN {X 0,Y 312.536,Z 149.552,A -85,B 0,C 180,E1 -15442.617,E2 -15442.617} C_VEL
LIN {X 0,Y 312.518,Z 149.555,A -85,B 0,C 180,E1 -15446.311,E2 -15446.311} C_VEL
LIN {X 0,Y 312.543,Z 149.549,A -85,B 0,C 180,E1 -15450.35,E2 -15450.35} C_VEL
LIN {X 0,Y 312.601,Z 149.546,A -85,B 0,C 180,E1 -15454.065,E2 -15454.065} C_VEL
LIN {X 0,Y 312.563,Z 149.552,A -85,B 0,C 180,E1 -15457.527,E2 -15457.527} C_VEL
LIN {X 0,Y 312.637,Z 149.54,A -85,B 0,C 180,E1 -15461.657,E2 -15461.657} C_VEL
LIN {X 0,Y 312.692,Z 149.535,A -85,B 0,C 180,E1 -15465.686,E2 -15465.686} C_VEL
LIN {X 0,Y 312.701,Z 149.533,A -85,B 0,C 180,E1 -15469.642,E2 -15469.642} C_VEL
LIN {X 0,Y 312.871,Z 149.508,A -85,B 0,C 180,E1 -15472.255,E2 -15472.255} C_VEL
LIN {X 0,Y 312.717,Z 149.528,A -85,B 0,C 180,E1 -15474.843,E2 -15474.843} C_VEL
LIN {X 0,Y 312.99,Z 149.496,A -85,B 0,C 180,E1 -15478.714,E2 -15478.714} C_VEL
LIN {X 0,Y 312.99,Z 149.497,A -85,B 0,C 180,E1 -15481.287,E2 -15481.287} C_VEL
LIN {X 0,Y 312.715,Z 149.532,A -85,B 0,C 180,E1 -15485.158,E2 -15485.158} C_VEL
LIN {X 0,Y 312.865,Z 149.51,A -85,B 0,C 180,E1 -15487.746,E2 -15487.746} C_VEL
LIN {X 0,Y 312.669,Z 149.533,A -85,B 0,C 180,E1 -15491.672,E2 -15491.672} C_VEL
LIN {X 0,Y 312.699,Z 149.535,A -85,B 0,C 180,E1 -15494.888,E2 -15494.888} C_VEL
LIN {X 0,Y 312.629,Z 149.539,A -85,B 0,C 180,E1 -15499.236,E2 -15499.236} C_VEL
LIN {X 0,Y 312.526,Z 149.556,A -85,B 0,C 180,E1 -15502.781,E2 -15502.781} C_VEL
LIN {X 0,Y 312.602,Z 149.544,A -85,B 0,C 180,E1 -15505.936,E2 -15505.936} C_VEL
LIN {X 0,Y 312.545,Z 149.551,A -85,B 0,C 180,E1 -15509.65,E2 -15509.65} C_VEL
LIN {X 0,Y 312.519,Z 149.554,A -85,B 0,C 180,E1 -15513.689,E2 -15513.689} C_VEL
LIN {X 0,Y 312.541,Z 149.551,A -85,B 0,C 180,E1 -15517.383,E2 -15517.383} C_VEL
LIN {X 0,Y 312.5,Z 149.557,A -85,B 0,C 180,E1 -15520.708,E2 -15520.708} C_VEL
LIN {X 0,Y 312.469,Z 149.563,A -85,B 0,C 180,E1 -15524.207,E2 -15524.207} C_VEL
LIN {X 0,Y 312.527,Z 149.558,A -85,B 0,C 180,E1 -15527.911,E2 -15527.911} C_VEL
LIN {X 0,Y 312.558,Z 149.554,A -85,B 0,C 180,E1 -15531.906,E2 -15531.906} C_VEL
LIN {X 0,Y 312.508,Z 149.559,A -85,B 0,C 180,E1 -15535.79,E2 -15535.79} C_VEL
LIN {X 0,Y 312.551,Z 149.609,A -85,B 0,C 180,E1 -15536.866,E2 -15536.866} C_VEL
LIN {X 0,Y 315.496,Z 163.066,A -85,B 0,C 180,E1 -15540.655,E2 -15540.655} C_VEL
LIN {X 0,Y 316.86,Z 169.974,A -85,B 0,C 180,E1 -15542.525,E2 -15542.525} C_VEL
LIN {X 0,Y 317.009,Z 173.187,A -85,B 0,C 180,E1 -15543.349,E2 -15543.349} C_VEL
LIN {X 0,Y 316.015,Z 181.418,A -85,B 0,C 180,E1 -15545.362,E2 -15545.362} C_VEL
LIN {X 0,Y 320.767,Z 216.246,A -85,B 0,C 180,E1 -15546.578,E2 -15546.578} C_VEL
LIN {X 0,Y 321.964,Z 226.415,A -85,B 0,C 180,E1 -15546.912,E2 -15546.912} C_VEL
LIN {X 0,Y 320.361,Z 291.241,A -85,B 0,C 180,E1 -15548.483,E2 -15548.483} C_VEL
LIN {X 0,Y 319.544,Z 304.659,A -85,B 0,C 180,E1 -15549.059,E2 -15549.059} C_VEL
LIN {X 0,Y 318.501,Z 316.938,A -85,B 0,C 180,E1 -15549.832,E2 -15549.832} C_VEL
LIN {X 0,Y 317.348,Z 327.999,A -85,B 0,C 180,E1 -15550.766,E2 -15550.766} C_VEL
LIN {X 0,Y 315.926,Z 339.577,A -85,B 0,C 180,E1 -15552.022,E2 -15552.022} C_VEL
LIN {X 0,Y 314.701,Z 350.055,A -85,B 0,C 180,E1 -15553.457,E2 -15553.457} C_VEL
LIN {X 0,Y 313.614,Z 359.465,A -85,B 0,C 180,E1 -15555.066,E2 -15555.066} C_VEL
LIN {X 0,Y 312.502,Z 368.574,A -85,B 0,C 180,E1 -15557.003,E2 -15557.003} C_VEL
LIN {X 0,Y 311.618,Z 375.894,A -85,B 0,C 180,E1 -15558.948,E2 -15558.948} C_VEL
LIN {X 0,Y 311.151,Z 381.73,A -85,B 0,C 180,E1 -15560.903,E2 -15560.903} C_VEL
LIN {X 0,Y 310.904,Z 386.3,A -85,B 0,C 180,E1 -15562.858,E2 -15562.858} C_VEL
LIN {X 0,Y 310.798,Z 389.746,A -85,B 0,C 180,E1 -15564.81,E2 -15564.81} C_VEL
LIN {X 0,Y 310.844,Z 391.447,A -85,B 0,C 180,E1 -15566.111,E2 -15566.111} C_VEL
LIN {X 0,Y 310.92,Z 393.596,A -85,B 0,C 180,E1 -15568.705,E2 -15568.705} C_VEL
LIN {X 0,Y 310.992,Z 394.019,A -85,B 0,C 180,E1 -15570,E2 -15570} C_VEL
LIN {X 0,Y 310.873,Z 394.012,A -85,B 0,C 180,E1 -15571.295,E2 -15571.295} C_VEL
LIN {X 0,Y 310.796,Z 392.816,A -85,B 0,C 180,E1 -15573.89,E2 -15573.89} C_VEL
LIN {X 0,Y 310.724,Z 391.067,A -85,B 0,C 180,E1 -15575.614,E2 -15575.614} C_VEL
LIN {X 0,Y 310.958,Z 387.82,A -85,B 0,C 180,E1 -15577.794,E2 -15577.794} C_VEL
LIN {X 0,Y 311.321,Z 383.806,A -85,B 0,C 180,E1 -15579.748,E2 -15579.748} C_VEL
LIN {X 0,Y 312.145,Z 377.694,A -85,B 0,C 180,E1 -15582.021,E2 -15582.021} C_VEL
LIN {X 0,Y 313.299,Z 371.006,A -85,B 0,C 180,E1 -15583.954,E2 -15583.954} C_VEL
LIN {X 0,Y 314.651,Z 362.915,A -85,B 0,C 180,E1 -15585.839,E2 -15585.839} C_VEL
LIN {X 0,Y 315.988,Z 354.316,A -85,B 0,C 180,E1 -15587.473,E2 -15587.473} C_VEL
LIN {X 0,Y 317.698,Z 344.039,A -85,B 0,C 180,E1 -15589.044,E2 -15589.044} C_VEL
LIN {X 0,Y 319.576,Z 332.476,A -85,B 0,C 180,E1 -15590.433,E2 -15590.433} C_VEL
LIN {X 0,Y 321.165,Z 321.182,A -85,B 0,C 180,E1 -15591.502,E2 -15591.502} C_VEL
LIN {X 0,Y 322.651,Z 308.519,A -85,B 0,C 180,E1 -15592.407,E2 -15592.407} C_VEL
LIN {X 0,Y 323.914,Z 294.53,A -85,B 0,C 180,E1 -15593.105,E2 -15593.105} C_VEL
LIN {X 0,Y 324.577,Z 281.063,A -85,B 0,C 180,E1 -15593.521,E2 -15593.521} C_VEL
LIN {X 0,Y 326.139,Z 225.517,A -85,B 0,C 180,E1 -15594.867,E2 -15594.867} C_VEL
LIN {X 0,Y 323.048,Z 203.393,A -85,B 0,C 180,E1 -15595.78,E2 -15595.78} C_VEL
LIN {X 0,Y 318.876,Z 181.689,A -85,B 0,C 180,E1 -15596.83,E2 -15596.83} C_VEL
LIN {X 0,Y 318.289,Z 178.71,A -85,B 0,C 180,E1 -15597.015,E2 -15597.015} C_VEL
LIN {X 0,Y 318.608,Z 176.376,A -85,B 0,C 180,E1 -15597.595,E2 -15597.595} C_VEL
LIN {X 0,Y 317.191,Z 168.418,A -85,B 0,C 180,E1 -15599.864,E2 -15599.864} C_VEL
LIN {X 0,Y 314.647,Z 157.559,A -85,B 0,C 180,E1 -15603.177,E2 -15603.177} C_VEL
LIN {X 0,Y 312.532,Z 149.559,A -85,B 0,C 180,E1 -15605.835,E2 -15605.835} C_VEL
LIN {X 0,Y 312.536,Z 149.558,A -85,B 0,C 180,E1 -15609.023,E2 -15609.023} C_VEL
LIN {X 0,Y 312.526,Z 149.561,A -85,B 0,C 180,E1 -15612.425,E2 -15612.425} C_VEL
LIN {X 0,Y 312.482,Z 149.562,A -85,B 0,C 180,E1 -15616.03,E2 -15616.03} C_VEL
LIN {X 0,Y 312.5,Z 149.559,A -85,B 0,C 180,E1 -15619.292,E2 -15619.292} C_VEL
LIN {X 0,Y 312.552,Z 149.553,A -85,B 0,C 180,E1 -15622.618,E2 -15622.618} C_VEL
LIN {X 0,Y 312.519,Z 149.553,A -85,B 0,C 180,E1 -15626.311,E2 -15626.311} C_VEL
LIN {X 0,Y 312.544,Z 149.546,A -85,B 0,C 180,E1 -15630.35,E2 -15630.35} C_VEL
LIN {X 0,Y 312.602,Z 149.538,A -85,B 0,C 180,E1 -15634.064,E2 -15634.064} C_VEL
LIN {X 0,Y 312.563,Z 149.542,A -85,B 0,C 180,E1 -15637.527,E2 -15637.527} C_VEL
LIN {X 0,Y 312.637,Z 149.534,A -85,B 0,C 180,E1 -15641.656,E2 -15641.656} C_VEL
LIN {X 0,Y 312.692,Z 149.529,A -85,B 0,C 180,E1 -15645.686,E2 -15645.686} C_VEL
LIN {X 0,Y 312.701,Z 149.53,A -85,B 0,C 180,E1 -15649.642,E2 -15649.642} C_VEL
LIN {X 0,Y 312.871,Z 149.505,A -85,B 0,C 180,E1 -15652.254,E2 -15652.254} C_VEL
LIN {X 0,Y 312.716,Z 149.533,A -85,B 0,C 180,E1 -15654.842,E2 -15654.842} C_VEL
LIN {X 0,Y 312.989,Z 149.497,A -85,B 0,C 180,E1 -15658.713,E2 -15658.713} C_VEL
LIN {X 0,Y 312.989,Z 149.499,A -85,B 0,C 180,E1 -15661.286,E2 -15661.286} C_VEL
LIN {X 0,Y 312.714,Z 149.53,A -85,B 0,C 180,E1 -15665.157,E2 -15665.157} C_VEL
LIN {X 0,Y 312.851,Z 149.515,A -85,B 0,C 180,E1 -15667.746,E2 -15667.746} C_VEL
LIN {X 0,Y 312.667,Z 149.535,A -85,B 0,C 180,E1 -15671.671,E2 -15671.671} C_VEL
LIN {X 0,Y 312.698,Z 149.536,A -85,B 0,C 180,E1 -15674.887,E2 -15674.887} C_VEL
LIN {X 0,Y 312.629,Z 149.544,A -85,B 0,C 180,E1 -15679.237,E2 -15679.237} C_VEL
LIN {X 0,Y 312.544,Z 149.558,A -85,B 0,C 180,E1 -15682.789,E2 -15682.789} C_VEL
LIN {X 0,Y 312.576,Z 149.716,A -85,B 0,C 180,E1 -15684.845,E2 -15684.845} C_VEL
LIN {X 0,Y 313.141,Z 151.65,A -85,B 0,C 180,E1 -15685.503,E2 -15685.503} C_VEL
LIN {X 0,Y 320.841,Z 166.938,A -85,B 0,C 180,E1 -15686.826,E2 -15686.826} C_VEL
LIN {X 0,Y 327.003,Z 181.232,A -85,B 0,C 180,E1 -15687.869,E2 -15687.869} C_VEL
LIN {X 0,Y 327.463,Z 182.766,A -85,B 0,C 180,E1 -15687.957,E2 -15687.957} C_VEL
LIN {X 0,Y 324.983,Z 258.363,A -85,B 0,C 180,E1 -15689.804,E2 -15689.804} C_VEL
LIN {X 0,Y 324.224,Z 271.539,A -85,B 0,C 180,E1 -15690.374,E2 -15690.374} C_VEL
LIN {X 0,Y 323.254,Z 284.226,A -85,B 0,C 180,E1 -15691.185,E2 -15691.185} C_VEL
LIN {X 0,Y 322.021,Z 295.84,A -85,B 0,C 180,E1 -15692.186,E2 -15692.186} C_VEL
LIN {X 0,Y 320.661,Z 306.375,A -85,B 0,C 180,E1 -15693.344,E2 -15693.344} C_VEL
LIN {X 0,Y 319.176,Z 316.324,A -85,B 0,C 180,E1 -15694.703,E2 -15694.703} C_VEL
LIN {X 0,Y 317.572,Z 325.692,A -85,B 0,C 180,E1 -15696.274,E2 -15696.274} C_VEL
LIN {X 0,Y 316.176,Z 333.35,A -85,B 0,C 180,E1 -15697.857,E2 -15697.857} C_VEL
LIN {X 0,Y 314.821,Z 340.35,A -85,B 0,C 180,E1 -15699.632,E2 -15699.632} C_VEL
LIN {X 0,Y 313.537,Z 347.138,A -85,B 0,C 180,E1 -15701.815,E2 -15701.815} C_VEL
LIN {X 0,Y 312.534,Z 352.3,A -85,B 0,C 180,E1 -15703.98,E2 -15703.98} C_VEL
LIN {X 0,Y 311.751,Z 356.099,A -85,B 0,C 180,E1 -15706.169,E2 -15706.169} C_VEL
LIN {X 0,Y 311.239,Z 358.465,A -85,B 0,C 180,E1 -15708.173,E2 -15708.173} C_VEL
LIN {X 0,Y 310.847,Z 360.023,A -85,B 0,C 180,E1 -15710.724,E2 -15710.724} C_VEL
LIN {X 0,Y 310.734,Z 360.231,A -85,B 0,C 180,E1 -15712.362,E2 -15712.362} C_VEL
LIN {X 0,Y 310.745,Z 359.512,A -85,B 0,C 180,E1 -15714.508,E2 -15714.508} C_VEL
LIN {X 0,Y 310.983,Z 357.582,A -85,B 0,C 180,E1 -15716.738,E2 -15716.738} C_VEL
LIN {X 0,Y 311.36,Z 354.248,A -85,B 0,C 180,E1 -15719.063,E2 -15719.063} C_VEL
LIN {X 0,Y 311.816,Z 350.504,A -85,B 0,C 180,E1 -15720.922,E2 -15720.922} C_VEL
LIN {X 0,Y 312.414,Z 345.37,A -85,B 0,C 180,E1 -15722.901,E2 -15722.901} C_VEL
LIN {X 0,Y 313.222,Z 339.263,A -85,B 0,C 180,E1 -15724.766,E2 -15724.766} C_VEL
LIN {X 0,Y 314.288,Z 331.11,A -85,B 0,C 180,E1 -15726.751,E2 -15726.751} C_VEL
LIN {X 0,Y 315.541,Z 321.422,A -85,B 0,C 180,E1 -15728.628,E2 -15728.628} C_VEL
LIN {X 0,Y 316.748,Z 311.102,A -85,B 0,C 180,E1 -15730.223,E2 -15730.223} C_VEL
LIN {X 0,Y 317.961,Z 300.095,A -85,B 0,C 180,E1 -15731.574,E2 -15731.574} C_VEL
LIN {X 0,Y 319.111,Z 287.502,A -85,B 0,C 180,E1 -15732.786,E2 -15732.786} C_VEL
LIN {X 0,Y 319.869,Z 275.872,A -85,B 0,C 180,E1 -15733.632,E2 -15733.632} C_VEL
LIN {X 0,Y 320.598,Z 262.726,A -85,B 0,C 180,E1 -15734.314,E2 -15734.314} C_VEL
LIN {X 0,Y 321.07,Z 249.179,A -85,B 0,C 180,E1 -15734.748,E2 -15734.748} C_VEL
LIN {X 0,Y 322.843,Z 178.025,A -85,B 0,C 180,E1 -15736.426,E2 -15736.426} C_VEL
LIN {X 0,Y 318.851,Z 165.928,A -85,B 0,C 180,E1 -15737.004,E2 -15737.004} C_VEL
LIN {X 0,Y 313.443,Z 151.974,A -85,B 0,C 180,E1 -15737.749,E2 -15737.749} C_VEL
LIN {X 0,Y 312.672,Z 149.54,A -85,B 0,C 180,E1 -15737.877,E2 -15737.877} C_VEL
LIN {X 0,Y 312.856,Z 149.513,A -85,B 0,C 180,E1 -15742.254,E2 -15742.254} C_VEL
LIN {X 0,Y 312.714,Z 149.531,A -85,B 0,C 180,E1 -15744.842,E2 -15744.842} C_VEL
LIN {X 0,Y 312.988,Z 149.496,A -85,B 0,C 180,E1 -15748.713,E2 -15748.713} C_VEL
LIN {X 0,Y 312.988,Z 149.501,A -85,B 0,C 180,E1 -15751.287,E2 -15751.287} C_VEL
LIN {X 0,Y 312.706,Z 149.536,A -85,B 0,C 180,E1 -15755.158,E2 -15755.158} C_VEL
LIN {X 0,Y 312.799,Z 149.52,A -85,B 0,C 180,E1 -15757.748,E2 -15757.748} C_VEL
LIN {X 0,Y 312.663,Z 149.537,A -85,B 0,C 180,E1 -15761.672,E2 -15761.672} C_VEL
LIN {X 0,Y 312.667,Z 149.54,A -85,B 0,C 180,E1 -15764.865,E2 -15764.865} C_VEL
LIN {X 0,Y 312.585,Z 149.548,A -85,B 0,C 180,E1 -15769.213,E2 -15769.213} C_VEL
LIN {X 0,Y 312.526,Z 149.558,A -85,B 0,C 180,E1 -15772.781,E2 -15772.781} C_VEL
LIN {X 0,Y 312.582,Z 149.55,A -85,B 0,C 180,E1 -15776.723,E2 -15776.723} C_VEL
LIN {X 0,Y 312.544,Z 149.55,A -85,B 0,C 180,E1 -15779.65,E2 -15779.65} C_VEL
LIN {X 0,Y 312.518,Z 149.554,A -85,B 0,C 180,E1 -15783.689,E2 -15783.689} C_VEL
LIN {X 0,Y 312.524,Z 149.553,A -85,B 0,C 180,E1 -15787.385,E2 -15787.385} C_VEL
LIN {X 0,Y 312.488,Z 149.558,A -85,B 0,C 180,E1 -15790.709,E2 -15790.709} C_VEL
LIN {X 0,Y 312.45,Z 149.567,A -85,B 0,C 180,E1 -15794.21,E2 -15794.21} C_VEL
LIN {X 0,Y 312.432,Z 149.564,A -85,B 0,C 180,E1 -15795.491,E2 -15795.491} C_VEL
LIN {X 0,Y 311.799,Z 149.647,A -85,B 0,C 180,E1 -15796.568,E2 -15796.568} C_VEL
LIN {X 0,Y 308.943,Z 150.001,A -85,B 0,C 180,E1 -15798.32,E2 -15798.32} C_VEL
LIN {X 0,Y 306.52,Z 150.301,A -85,B 0,C 180,E1 -15799.741,E2 -15799.741} C_VEL
LIN {X 0,Y 305.512,Z 150.424,A -85,B 0,C 180,E1 -15800.842,E2 -15800.842} C_VEL
LIN {X 0,Y 305.448,Z 150.431,A -85,B 0,C 180,E1 -15801.215,E2 -15801.215} C_VEL
LIN {X 0,Y 305.461,Z 150.432,A -85,B 0,C 180,E1 -15804.887,E2 -15804.887} C_VEL
LIN {X 0,Y 305.451,Z 150.434,A -85,B 0,C 180,E1 -15808.355,E2 -15808.355} C_VEL
LIN {X 0,Y 305.519,Z 150.422,A -85,B 0,C 180,E1 -15811.114,E2 -15811.114} C_VEL
LIN {X 0,Y 305.57,Z 150.421,A -85,B 0,C 180,E1 -15814.088,E2 -15814.088} C_VEL
LIN {X 0,Y 305.48,Z 150.43,A -85,B 0,C 180,E1 -15818.402,E2 -15818.402} C_VEL
LIN {X 0,Y 305.588,Z 150.417,A -85,B 0,C 180,E1 -15821.218,E2 -15821.218} C_VEL
LIN {X 0,Y 305.648,Z 150.412,A -85,B 0,C 180,E1 -15825.349,E2 -15825.349} C_VEL
LIN {X 0,Y 305.638,Z 150.415,A -85,B 0,C 180,E1 -15829.4,E2 -15829.4} C_VEL
LIN {X 0,Y 305.812,Z 150.387,A -85,B 0,C 180,E1 -15832.075,E2 -15832.075} C_VEL
LIN {X 0,Y 305.688,Z 150.403,A -85,B 0,C 180,E1 -15834.724,E2 -15834.724} C_VEL
LIN {X 0,Y 305.956,Z 150.372,A -85,B 0,C 180,E1 -15838.684,E2 -15838.684} C_VEL
LIN {X 0,Y 305.956,Z 150.372,A -85,B 0,C 180,E1 -15841.317,E2 -15841.317} C_VEL
LIN {X 0,Y 305.845,Z 150.386,A -85,B 0,C 180,E1 -15846.598,E2 -15846.598} C_VEL
LIN {X 0,Y 305.735,Z 150.4,A -85,B 0,C 180,E1 -15849.26,E2 -15849.26} C_VEL
LIN {X 0,Y 305.588,Z 150.417,A -85,B 0,C 180,E1 -15853.296,E2 -15853.296} C_VEL
LIN {X 0,Y 305.593,Z 150.417,A -85,B 0,C 180,E1 -15856.02,E2 -15856.02} C_VEL
LIN {X 0,Y 305.575,Z 150.417,A -85,B 0,C 180,E1 -15859.445,E2 -15859.445} C_VEL
LIN {X 0,Y 305.486,Z 150.431,A -85,B 0,C 180,E1 -15863.04,E2 -15863.04} C_VEL
LIN {X 0,Y 305.547,Z 150.425,A -85,B 0,C 180,E1 -15866.227,E2 -15866.227} C_VEL
LIN {X 0,Y 305.495,Z 150.429,A -85,B 0,C 180,E1 -15869.05,E2 -15869.05} C_VEL
LIN {X 0,Y 305.465,Z 150.433,A -85,B 0,C 180,E1 -15873.517,E2 -15873.517} C_VEL
LIN {X 0,Y 305.498,Z 150.429,A -85,B 0,C 180,E1 -15876.737,E2 -15876.737} C_VEL
LIN {X 0,Y 305.466,Z 150.437,A -85,B 0,C 180,E1 -15880.107,E2 -15880.107} C_VEL
LIN {X 0,Y 305.447,Z 150.437,A -85,B 0,C 180,E1 -15883.652,E2 -15883.652} C_VEL
LIN {X 0,Y 305.486,Z 150.431,A -85,B 0,C 180,E1 -15887.408,E2 -15887.408} C_VEL
LIN {X 0,Y 305.519,Z 150.43,A -85,B 0,C 180,E1 -15891.604,E2 -15891.604} C_VEL
LIN {X 0,Y 305.464,Z 150.434,A -85,B 0,C 180,E1 -15894.887,E2 -15894.887} C_VEL
LIN {X 0,Y 305.496,Z 150.526,A -85,B 0,C 180,E1 -15896.487,E2 -15896.487} C_VEL
LIN {X 0,Y 308.371,Z 163.627,A -85,B 0,C 180,E1 -15900.273,E2 -15900.273} C_VEL
LIN {X 0,Y 310.037,Z 172.187,A -85,B 0,C 180,E1 -15902.639,E2 -15902.639} C_VEL
